discrete alarms
   1: '1UZ1 (A01590) - Привід: перевищено інтервал технічного обслуговування двигуна', class WarningLiftUp, trigger "AlarmsWord1" bit 0
   2: '1UZ1 (A01666) - SI Motion P1 (CU): Постійний сигнал «1» на F-DI для безпечного квитування', class WarningLiftUp, trigger "AlarmsWord1" bit 1
   3: '1UZ1 (A01698) - SI P1 (CU): Активний режим введення в експлуатацію', class WarningLiftUp, trigger "AlarmsWord1" bit 2
   4: '1UZ1 (A01699) - SI P1 (CU): Потрібна тестова зупинка для STO', class WarningLiftUp, trigger "AlarmsWord1" bit 3
   5: '1UZ1 (A01900) - PB/PN: Конфігурація Помилка телеграми', class WarningLiftUp, trigger "AlarmsWord1" bit 4
   6: '1UZ1(A01920) - PROFIBUS: перервано циклічне з’єднання', class WarningLiftUp, trigger "AlarmsWord1" bit 5
   7: '1UZ1 (A05000) - Силовий модуль: перегрів радіатора інвертора AC', class WarningLiftUp, trigger "AlarmsWord1" bit 6
   8: '1UZ1 (A05001) - Силовий модуль: перегрів кристала запірного шару', class WarningLiftUp, trigger "AlarmsWord1" bit 7
   9: '1UZ1 (A05002) - Силовий модуль: перегрів повітря на вході', class WarningLiftUp, trigger "AlarmsWord1" bit 8
   10: '1UZ1 (A05004) - Силовий модуль: перегрів випрямляча', class WarningLiftUp, trigger "AlarmsWord1" bit 9
   11: '1UZ1 (A05006) - Силовий модуль: перегрів за тепловою моделлю', class WarningLiftUp, trigger "AlarmsWord1" bit 10
   12: '1UZ1 (A07012) - Привід: Двигун температура модель 1/3 перегрів', class WarningLiftUp, trigger "AlarmsWord1" bit 11
   13: '1UZ1 (A01013) - CU: Досягнуто або перевищено граничний ресурс вентилятора', class WarningLiftUp, trigger "AlarmsWord1" bit 12
   14: '1UZ1 (A07321) - Привід: Автоматичний перезапуск активний', class WarningLiftUp, trigger "AlarmsWord1" bit 13
   15: '1UZ1 (A07400) - Привід: активний регулятор максимальної напруги кола постійного струму', class WarningLiftUp, trigger "AlarmsWord1" bit 14
   16: '1UZ1 (A07409) - Привід: керування U/f, активний регулятор обмеження струму', class WarningLiftUp, trigger "AlarmsWord1" bit 15
   18: '1UZ1 (A07805) - Ввід: перевантаження I²t силового модуля', class WarningLiftUp, trigger "AlarmsWord2" bit 0
   19: '1UZ1 (A07850) - Зовнішній аварійне повідомлення 1', class WarningLiftUp, trigger "AlarmsWord2" bit 1
   20: '1UZ1 (A07851) - Зовнішній аварійне повідомлення 2', class WarningLiftUp, trigger "AlarmsWord2" bit 2
   21: '1UZ1 (A07852) - Зовнішній аварійне повідомлення 3', class WarningLiftUp, trigger "AlarmsWord2" bit 3
   22: '1UZ1 (A07903) - Привід: відхилення швидкості двигуна', class WarningLiftUp, trigger "AlarmsWord2" bit 4
   23: '1UZ1 (A07910) - Привід: перегрів двигуна', class WarningLiftUp, trigger "AlarmsWord2" bit 5
   24: '1UZ1 (A07920) - Привід: крутний момент/швидкість занадто низькі', class WarningLiftUp, trigger "AlarmsWord2" bit 6
   25: '1UZ1 (A07921) - Привід: крутний момент/швидкість занадто високі', class WarningLiftUp, trigger "AlarmsWord2" bit 7
   26: '1UZ1 (A07922) - Привід: крутний момент/швидкість поза межами допуску', class WarningLiftUp, trigger "AlarmsWord2" bit 8
   27: '1UZ1 (A07927) - DC гальмівний активний', class WarningLiftUp, trigger "AlarmsWord2" bit 9
   28: '1UZ1 (A07980) - Привід: Обертовий вимірювання активовано', class WarningLiftUp, trigger "AlarmsWord2" bit 10
   29: '1UZ1 (A07981) - Привід: Увімкнути сигнали для обертовий вимірювання відсутній', class WarningLiftUp, trigger "AlarmsWord2" bit 11
   30: '1UZ1 (A07991) - Привід: Ідентифікація даних двигуна активовано', class WarningLiftUp, trigger "AlarmsWord2" bit 12
   31: '1UZ1 (A08511) - PN/COMM BOARD: Приймання конфігурація дані некоректний', class WarningLiftUp, trigger "AlarmsWord2" bit 13
   32: '1UZ1 (A08526) - PN/COMM BOARD: Відсутній циклічний з’єднання', class WarningLiftUp, trigger "AlarmsWord2" bit 14
   33: '1UZ1 (A08565) - PNCOMM BOARD: Узгодженість помилка що впливає на регульований параметри', class WarningLiftUp, trigger "AlarmsWord2" bit 15
   35: '1UZ1 (A30049) - Силовий модуль: несправний внутрішній вентилятор', class WarningLiftUp, trigger "AlarmsWord3" bit 0
   36: '1UZ1 (A30502) - Силовий модуль: Перенапруга кола постійного струму', class WarningLiftUp, trigger "AlarmsWord3" bit 1
   37: '1UZ1 (A30920) - Силовий модуль: несправність датчика температури', class WarningLiftUp, trigger "AlarmsWord3" bit 2
   39: '1UZ1 (F01000) - Внутрішня програмна помилка', class ErrorLiftUp, trigger "FaultsWord1" bit 0
   40: '1UZ1 (F01001) - Виняток операції з плаваючою комою', class ErrorLiftUp, trigger "FaultsWord1" bit 1
   41: '1UZ1 (F01015) - Внутрішня програмна помилка', class ErrorLiftUp, trigger "FaultsWord1" bit 2
   42: '1UZ1 (F01033) - Перемикання одиниць: некоректне опорне значення параметра', class ErrorLiftUp, trigger "FaultsWord1" bit 3
   43: '1UZ1 (F01034) - Перемикання одиниць: не вдалося обчислити значення параметрів після зміни опорного значення', class ErrorLiftUp, trigger "FaultsWord1" bit 4
   44: '1UZ1 (F01040) - Збережіть налаштування параметрів і виконайте повторне увімкнення живлення', class ErrorLiftUp, trigger "FaultsWord1" bit 5
   45: '1UZ1 (F01044) - CU: Помилка описових даних', class ErrorLiftUp, trigger "FaultsWord1" bit 6
   46: '1UZ1 (F01054) - CU: Перевищено системне обмеження', class ErrorLiftUp, trigger "FaultsWord1" bit 7
   47: '1UZ1 (F01105) - CU: Недостатньо пам’яті', class ErrorLiftUp, trigger "FaultsWord1" bit 8
   48: '1UZ1 (F01122) - Частота на вході вимірювального щупа занадто висока', class ErrorLiftUp, trigger "FaultsWord1" bit 9
   49: '1UZ1 (F01205) - CU: Переповнення часового кванта', class ErrorLiftUp, trigger "FaultsWord1" bit 10
   50: '1UZ1 (F01250) - CU: Некоректні дані CU-EEPROM, доступні лише для читання', class ErrorLiftUp, trigger "FaultsWord1" bit 11
   51: '1UZ1 (F01512) - BICO: масштабування недоступне', class ErrorLiftUp, trigger "FaultsWord1" bit 12
   52: '1UZ1 (F01600) - SI P1 (CU): Ініційовано зупинку A', class ErrorLiftUp, trigger "FaultsWord1" bit 13
   53: '1UZ1 (F01625) - SI P1 (CU): Помилка сигналу справності в даних безпеки', class ErrorLiftUp, trigger "FaultsWord1" bit 14
   54: '1UZ1 (F01650) - SI P1 (CU): Потрібне приймальне випробування', class ErrorLiftUp, trigger "FaultsWord1" bit 15
   56: '1UZ1 (F01659) - SI P1 (CU): Запит на запис параметра відхилено', class ErrorLiftUp, trigger "FaultsWord2" bit 0
   57: '1UZ1 (F01666) - SI Motion P1 (CU): Постійний сигнал «1» на F-DI для безпечного квитування', class ErrorLiftUp, trigger "FaultsWord2" bit 1
   58: '1UZ1 (F01910) - Польова шина: тайм-аут заданого значення', class ErrorLiftUp, trigger "FaultsWord2" bit 2
   59: '1UZ1 (F06310) - Ввід: напругу живлення (p0210) параметризовано некоректно', class ErrorLiftUp, trigger "FaultsWord2" bit 3
   60: '1UZ1 (F07011) - Привід: перегрів двигуна', class ErrorLiftUp, trigger "FaultsWord2" bit 4
   61: '1UZ1 (F07016) - Привід: Несправність датчика температури двигуна', class ErrorLiftUp, trigger "FaultsWord2" bit 5
   62: '1UZ1 (F07086) - Перемикання одиниць: порушення обмеження параметра через зміну опорного значення', class ErrorLiftUp, trigger "FaultsWord2" bit 6
   63: '1UZ1 (F07088) - Перемикання одиниць: порушення обмеження параметра через перемикання одиниць', class ErrorLiftUp, trigger "FaultsWord2" bit 7
   64: '1UZ1 (F07320) - Привід: Автоматичний перезапуск перервано', class ErrorLiftUp, trigger "FaultsWord2" bit 8
   65: '1UZ1 (F07330) - Підхоплення обертового двигуна: виміряний пошуковий струм занадто малий', class ErrorLiftUp, trigger "FaultsWord2" bit 9
   66: '1UZ1 (F07426) - Технологія регулятор фактичний значення обмежений', class ErrorLiftUp, trigger "FaultsWord2" bit 10
   67: '1UZ1 (F07801) - Привід: Двигун Перевищення струму', class ErrorLiftUp, trigger "FaultsWord2" bit 11
   68: '1UZ1 (F07807) - Привід: виявлено коротке замикання/замикання на землю', class ErrorLiftUp, trigger "FaultsWord2" bit 12
   69: '1UZ1 (F07860) - Зовнішній несправність 1', class ErrorLiftUp, trigger "FaultsWord2" bit 13
   70: '1UZ1 (F07861) - Зовнішній несправність 2', class ErrorLiftUp, trigger "FaultsWord2" bit 14
   71: '1UZ1 (F07862) - Зовнішній несправність 3', class ErrorLiftUp, trigger "FaultsWord2" bit 15
   74: '1UZ1 (F07900) - Привід: заклинювання двигуна/регулятор швидкості на межі', class ErrorLiftUp, trigger "FaultsWord3" bit 0
   75: '1UZ1 (F07901) - Привід: перевищення швидкості двигуна', class ErrorLiftUp, trigger "FaultsWord3" bit 1
   76: '1UZ1 (F07902) - Привід: двигун зупинився', class ErrorLiftUp, trigger "FaultsWord3" bit 2
   77: '1UZ1 (F07923) - Привід: крутний момент/швидкість занадто низькі', class ErrorLiftUp, trigger "FaultsWord3" bit 3
   78: '1UZ1 (F07924) - Привід: крутний момент/швидкість занадто високі', class ErrorLiftUp, trigger "FaultsWord3" bit 4
   79: '1UZ1 (F08501) - PN/COMM BOARD: тайм-аут заданого значення', class ErrorLiftUp, trigger "FaultsWord3" bit 5
   80: '1UZ1 (F08502) - PN/COMM BOARD: закінчився контрольний час сигналу справності', class ErrorLiftUp, trigger "FaultsWord3" bit 6
   81: '1UZ1 (F06210) - Ввід: Сумування струм занадто високий', class ErrorLiftUp, trigger "FaultsWord3" bit 7
   82: '1UZ1 (F13100) - Захист ноу-хау: помилка захисту від копіювання', class ErrorLiftUp, trigger "FaultsWord3" bit 8
   83: '1UZ1 (F13101) - Захист ноу-хау: неможливо активувати захист від копіювання', class ErrorLiftUp, trigger "FaultsWord3" bit 9
   84: '1UZ1 (F30001) - Силовий модуль: перевищення струму', class ErrorLiftUp, trigger "FaultsWord3" bit 10
   85: '1UZ1 (F30002) - Силовий модуль: перенапруга кола постійного струму', class ErrorLiftUp, trigger "FaultsWord3" bit 11
   86: '1UZ1 (F30003) - Силовий модуль: занижена напруга кола постійного струму', class ErrorLiftUp, trigger "FaultsWord3" bit 12
   87: '1UZ1 (F30004) - Силовий модуль: перегрів радіатора інвертора AC', class ErrorLiftUp, trigger "FaultsWord3" bit 13
   88: '1UZ1 (F30005) - Силовий модуль: перевантаження I²t', class ErrorLiftUp, trigger "FaultsWord3" bit 14
   89: '1UZ1 (F30011) - Силовий модуль: відсутня фаза мережі в головному колі', class ErrorLiftUp, trigger "FaultsWord3" bit 15
   91: '1UZ1 (F30015) - Силовий модуль: відсутня фаза кабелю двигуна', class ErrorLiftUp, trigger "FaultsWord4" bit 0
   92: '1UZ1 (F30021) - Силовий модуль: замикання на землю', class ErrorLiftUp, trigger "FaultsWord4" bit 1
   93: '1UZ1 (F30022) - Силовий модуль: контроль Uce', class ErrorLiftUp, trigger "FaultsWord4" bit 2
   94: '1UZ1 (F30027) - Силовий модуль: контроль часу попереднього заряду кола постійного струму', class ErrorLiftUp, trigger "FaultsWord4" bit 3
   95: '1UZ1 (F30035) - Силовий модуль: перегрів повітря на вході', class ErrorLiftUp, trigger "FaultsWord4" bit 4
   96: '1UZ1 (F30036) - Силовий модуль: внутрішній перегрів', class ErrorLiftUp, trigger "FaultsWord4" bit 5
   97: '1UZ1 (F30037) - Силовий модуль: перегрів випрямляча', class ErrorLiftUp, trigger "FaultsWord4" bit 6
   98: '1UZ1 (F30052) - Помилка даних EEPROM', class ErrorLiftUp, trigger "FaultsWord4" bit 7
   99: '1UZ1 (F30053) - FPGA дані несправний', class ErrorLiftUp, trigger "FaultsWord4" bit 8
   100: '1UZ1 (F30059) - Силовий модуль: несправний внутрішній вентилятор', class ErrorLiftUp, trigger "FaultsWord4" bit 9
   101: '1UZ1 (F30074) - Помилка зв’язку між Керування Модуль та Силовий модуль', class ErrorLiftUp, trigger "FaultsWord4" bit 10
   102: '1UZ1 (F30600) - SI P2: Ініційовано зупинку A', class ErrorLiftUp, trigger "FaultsWord4" bit 11
   103: '1UZ1 (F30664) - Помилка під час завантаження', class ErrorLiftUp, trigger "FaultsWord4" bit 12
   104: '1UZ1 (F30850) - Силовий модуль: Внутрішня програмна помилка', class ErrorLiftUp, trigger "FaultsWord4" bit 13
   38: '1UZ1 (F06211) - Ввід: сумарний струм неприпустимо високий', class ErrorLiftUp, trigger "FaultsWord4" bit 14
   105: '1UZ1 (F08510) - PN/COMM BOARD: некоректні дані конфігурації передавання', class ErrorLiftUp, trigger "FaultsWord4" bit 15
   106: '3UZ1 (A01590) - Привід: перевищено інтервал технічного обслуговування двигуна', class WarningTrolley, trigger "AlarmsWord1" bit 0
   107: '3UZ1 (A01666) - SI Motion P1 (CU): Постійний сигнал «1» на F-DI для безпечного квитування', class WarningTrolley, trigger "AlarmsWord1" bit 1
   108: '3UZ1 (A01698) - SI P1 (CU): Активний режим введення в експлуатацію', class WarningTrolley, trigger "AlarmsWord1" bit 2
   109: '3UZ1 (A01699) - SI P1 (CU): Потрібна тестова зупинка для STO', class WarningTrolley, trigger "AlarmsWord1" bit 3
   110: '3UZ1 (A01900) - PB/PN: Конфігурація Помилка телеграми', class WarningTrolley, trigger "AlarmsWord1" bit 4
   111: '3UZ1(A01920) - PROFIBUS: перервано циклічне з’єднання', class WarningTrolley, trigger "AlarmsWord1" bit 5
   112: '3UZ1 (A05000) - Силовий модуль: перегрів радіатора інвертора AC', class WarningTrolley, trigger "AlarmsWord1" bit 6
   113: '3UZ1 (A05001) - Силовий модуль: перегрів кристала запірного шару', class WarningTrolley, trigger "AlarmsWord1" bit 7
   114: '3UZ1 (A05002) - Силовий модуль: перегрів повітря на вході', class WarningTrolley, trigger "AlarmsWord1" bit 8
   115: '3UZ1 (A05004) - Силовий модуль: перегрів випрямляча', class WarningTrolley, trigger "AlarmsWord1" bit 9
   116: '3UZ1 (A05006) - Силовий модуль: перегрів за тепловою моделлю', class WarningTrolley, trigger "AlarmsWord1" bit 10
   117: '3UZ1 (A07012) - Привід: Двигун температура модель 1/3 перегрів', class WarningTrolley, trigger "AlarmsWord1" bit 11
   118: '3UZ1 (A01013) - CU: Досягнуто або перевищено граничний ресурс вентилятора', class WarningTrolley, trigger "AlarmsWord1" bit 12
   119: '3UZ1 (A07321) - Привід: Автоматичний перезапуск активний', class WarningTrolley, trigger "AlarmsWord1" bit 13
   120: '3UZ1 (A07400) - Привід: активний регулятор максимальної напруги кола постійного струму', class WarningTrolley, trigger "AlarmsWord1" bit 14
   121: '3UZ1 (A07409) - Привід: керування U/f, активний регулятор обмеження струму', class WarningTrolley, trigger "AlarmsWord1" bit 15
   122: '3UZ1 (A07805) - Ввід: перевантаження I²t силового модуля', class WarningTrolley, trigger "AlarmsWord2" bit 0
   123: '3UZ1 (A07850) - Зовнішній аварійне повідомлення 1', class WarningTrolley, trigger "AlarmsWord2" bit 1
   124: '3UZ1 (A07851) - Зовнішній аварійне повідомлення 2', class WarningTrolley, trigger "AlarmsWord2" bit 2
   125: '3UZ1 (A07852) - Зовнішній аварійне повідомлення 3', class WarningTrolley, trigger "AlarmsWord2" bit 3
   126: '3UZ1 (A07903) - Привід: відхилення швидкості двигуна', class WarningTrolley, trigger "AlarmsWord2" bit 4
   127: '3UZ1 (A07910) - Привід: перегрів двигуна', class WarningTrolley, trigger "AlarmsWord2" bit 5
   128: '3UZ1 (A07920) - Привід: крутний момент/швидкість занадто низькі', class WarningTrolley, trigger "AlarmsWord2" bit 6
   129: '3UZ1 (A07921) - Привід: крутний момент/швидкість занадто високі', class WarningTrolley, trigger "AlarmsWord2" bit 7
   130: '3UZ1 (A07922) - Привід: крутний момент/швидкість поза межами допуску', class WarningTrolley, trigger "AlarmsWord2" bit 8
   131: '3UZ1 (A07927) - DC гальмівний активний', class WarningTrolley, trigger "AlarmsWord2" bit 9
   132: '3UZ1 (A07980) - Привід: Обертовий вимірювання активовано', class WarningTrolley, trigger "AlarmsWord2" bit 10
   133: '3UZ1 (A07981) - Привід: Увімкнути сигнали для обертовий вимірювання відсутній', class WarningTrolley, trigger "AlarmsWord2" bit 11
   134: '3UZ1 (A07991) - Привід: Ідентифікація даних двигуна активовано', class WarningTrolley, trigger "AlarmsWord2" bit 12
   135: '3UZ1 (A08511) - PN/COMM BOARD: Приймання конфігурація дані некоректний', class WarningTrolley, trigger "AlarmsWord2" bit 13
   136: '3UZ1 (A08526) - PN/COMM BOARD: Відсутній циклічний з’єднання', class WarningTrolley, trigger "AlarmsWord2" bit 14
   137: '3UZ1 (A08565) - PNCOMM BOARD: Узгодженість помилка що впливає на регульований параметри', class WarningTrolley, trigger "AlarmsWord2" bit 15
   138: '3UZ1 (A30049) - Силовий модуль: несправний внутрішній вентилятор', class WarningTrolley, trigger "AlarmsWord3" bit 0
   139: '3UZ1 (A30502) - Силовий модуль: Перенапруга кола постійного струму', class WarningTrolley, trigger "AlarmsWord3" bit 1
   140: '3UZ1 (A30920) - Силовий модуль: несправність датчика температури', class WarningTrolley, trigger "AlarmsWord3" bit 2
   141: '3UZ1 (F01000) - Внутрішня програмна помилка', class ErrorTrolley, trigger "FaultsWord1" bit 0
   142: '3UZ1 (F01001) - Виняток операції з плаваючою комою', class ErrorTrolley, trigger "FaultsWord1" bit 1
   143: '3UZ1 (F01015) - Внутрішня програмна помилка', class ErrorTrolley, trigger "FaultsWord1" bit 2
   144: '3UZ1 (F01033) - Перемикання одиниць: некоректне опорне значення параметра', class ErrorTrolley, trigger "FaultsWord1" bit 3
   145: '3UZ1 (F01034) - Перемикання одиниць: не вдалося обчислити значення параметрів після зміни опорного значення', class ErrorTrolley, trigger "FaultsWord1" bit 4
   146: '3UZ1 (F01040) - Збережіть налаштування параметрів і виконайте повторне увімкнення живлення', class ErrorTrolley, trigger "FaultsWord1" bit 5
   147: '3UZ1 (F01044) - CU: Помилка описових даних', class ErrorTrolley, trigger "FaultsWord1" bit 6
   148: '3UZ1 (F01054) - CU: Перевищено системне обмеження', class ErrorTrolley, trigger "FaultsWord1" bit 7
   149: '3UZ1 (F01105) - CU: Недостатньо пам’яті', class ErrorTrolley, trigger "FaultsWord1" bit 8
   150: '3UZ1 (F01122) - Частота на вході вимірювального щупа занадто висока', class ErrorTrolley, trigger "FaultsWord1" bit 9
   151: '3UZ1 (F01205) - CU: Переповнення часового кванта', class ErrorTrolley, trigger "FaultsWord1" bit 10
   152: '3UZ1 (F01250) - CU: Некоректні дані CU-EEPROM, доступні лише для читання', class ErrorTrolley, trigger "FaultsWord1" bit 11
   153: '3UZ1 (F01512) - BICO: масштабування недоступне', class ErrorTrolley, trigger "FaultsWord1" bit 12
   154: '3UZ1 (F01600) - SI P1 (CU): Ініційовано зупинку A', class ErrorTrolley, trigger "FaultsWord1" bit 13
   155: '3UZ1 (F01625) - SI P1 (CU): Помилка сигналу справності в даних безпеки', class ErrorTrolley, trigger "FaultsWord1" bit 14
   156: '3UZ1 (F01650) - SI P1 (CU): Потрібне приймальне випробування', class ErrorTrolley, trigger "FaultsWord1" bit 15
   157: '3UZ1 (F01659) - SI P1 (CU): Запит на запис параметра відхилено', class ErrorTrolley, trigger "FaultsWord2" bit 0
   158: '3UZ1 (F01666) - SI Motion P1 (CU): Постійний сигнал «1» на F-DI для безпечного квитування', class ErrorTrolley, trigger "FaultsWord2" bit 1
   159: '3UZ1 (F01910) - Польова шина: тайм-аут заданого значення', class ErrorTrolley, trigger "FaultsWord2" bit 2
   160: '3UZ1 (F06310) - Ввід: напругу живлення (p0210) параметризовано некоректно', class ErrorTrolley, trigger "FaultsWord2" bit 3
   161: '3UZ1 (F07011) - Привід: перегрів двигуна', class ErrorTrolley, trigger "FaultsWord2" bit 4
   162: '3UZ1 (F07016) - Привід: Несправність датчика температури двигуна', class ErrorTrolley, trigger "FaultsWord2" bit 5
   163: '3UZ1 (F07086) - Перемикання одиниць: порушення обмеження параметра через зміну опорного значення', class ErrorTrolley, trigger "FaultsWord2" bit 6
   164: '3UZ1 (F07088) - Перемикання одиниць: порушення обмеження параметра через перемикання одиниць', class ErrorTrolley, trigger "FaultsWord2" bit 7
   165: '3UZ1 (F07320) - Привід: Автоматичний перезапуск перервано', class ErrorTrolley, trigger "FaultsWord2" bit 8
   166: '3UZ1 (F07330) - Підхоплення обертового двигуна: виміряний пошуковий струм занадто малий', class ErrorTrolley, trigger "FaultsWord2" bit 9
   167: '3UZ1 (F07426) - Технологія регулятор фактичний значення обмежений', class ErrorTrolley, trigger "FaultsWord2" bit 10
   168: '3UZ1 (F07801) - Привід: Двигун Перевищення струму', class ErrorTrolley, trigger "FaultsWord2" bit 11
   169: '3UZ1 (F07807) - Привід: виявлено коротке замикання/замикання на землю', class ErrorTrolley, trigger "FaultsWord2" bit 12
   170: '3UZ1 (F07860) - Зовнішній несправність 1', class ErrorTrolley, trigger "FaultsWord2" bit 13
   171: '3UZ1 (F07861) - Зовнішній несправність 2', class ErrorTrolley, trigger "FaultsWord2" bit 14
   172: '3UZ1 (F07862) - Зовнішній несправність 3', class ErrorTrolley, trigger "FaultsWord2" bit 15
   173: '3UZ1 (F07900) - Привід: заклинювання двигуна/регулятор швидкості на межі', class ErrorTrolley, trigger "FaultsWord3" bit 0
   174: '3UZ1 (F07901) - Привід: перевищення швидкості двигуна', class ErrorTrolley, trigger "FaultsWord3" bit 1
   175: '3UZ1 (F07902) - Привід: двигун зупинився', class ErrorTrolley, trigger "FaultsWord3" bit 2
   176: '3UZ1 (F07923) - Привід: крутний момент/швидкість занадто низькі', class ErrorTrolley, trigger "FaultsWord3" bit 3
   177: '3UZ1 (F07924) - Привід: крутний момент/швидкість занадто високі', class ErrorTrolley, trigger "FaultsWord3" bit 4
   178: '3UZ1 (F08501) - PN/COMM BOARD: тайм-аут заданого значення', class ErrorTrolley, trigger "FaultsWord3" bit 5
   179: '3UZ1 (F08502) - PN/COMM BOARD: закінчився контрольний час сигналу справності', class ErrorTrolley, trigger "FaultsWord3" bit 6
   180: '3UZ1 (F06210) - Ввід: Сумування струм занадто високий', class ErrorTrolley, trigger "FaultsWord3" bit 7
   181: '3UZ1 (F13100) - Захист ноу-хау: помилка захисту від копіювання', class ErrorTrolley, trigger "FaultsWord3" bit 8
   182: '3UZ1 (F13101) - Захист ноу-хау: неможливо активувати захист від копіювання', class ErrorTrolley, trigger "FaultsWord3" bit 9
   183: '3UZ1 (F30001) - Силовий модуль: перевищення струму', class ErrorTrolley, trigger "FaultsWord3" bit 10
   184: '3UZ1 (F30002) - Силовий модуль: перенапруга кола постійного струму', class ErrorTrolley, trigger "FaultsWord3" bit 11
   185: '3UZ1 (F30003) - Силовий модуль: занижена напруга кола постійного струму', class ErrorTrolley, trigger "FaultsWord3" bit 12
   186: '3UZ1 (F30004) - Силовий модуль: перегрів радіатора інвертора AC', class ErrorTrolley, trigger "FaultsWord3" bit 13
   187: '3UZ1 (F30005) - Силовий модуль: перевантаження I²t', class ErrorTrolley, trigger "FaultsWord3" bit 14
   188: '3UZ1 (F30011) - Силовий модуль: відсутня фаза мережі в головному колі', class ErrorTrolley, trigger "FaultsWord3" bit 15
   189: '3UZ1 (F30015) - Силовий модуль: відсутня фаза кабелю двигуна', class ErrorTrolley, trigger "FaultsWord4" bit 0
   190: '3UZ1 (F30021) - Силовий модуль: замикання на землю', class ErrorTrolley, trigger "FaultsWord4" bit 1
   191: '3UZ1 (F30022) - Силовий модуль: контроль Uce', class ErrorTrolley, trigger "FaultsWord4" bit 2
   192: '3UZ1 (F30027) - Силовий модуль: контроль часу попереднього заряду кола постійного струму', class ErrorTrolley, trigger "FaultsWord4" bit 3
   193: '3UZ1 (F30035) - Силовий модуль: перегрів повітря на вході', class ErrorTrolley, trigger "FaultsWord4" bit 4
   194: '3UZ1 (F30036) - Силовий модуль: внутрішній перегрів', class ErrorTrolley, trigger "FaultsWord4" bit 5
   195: '3UZ1 (F30037) - Силовий модуль: перегрів випрямляча', class ErrorTrolley, trigger "FaultsWord4" bit 6
   196: '3UZ1 (F30052) - Помилка даних EEPROM', class ErrorTrolley, trigger "FaultsWord4" bit 7
   197: '3UZ1 (F30053) - FPGA дані несправний', class ErrorTrolley, trigger "FaultsWord4" bit 8
   198: '3UZ1 (F30059) - Силовий модуль: несправний внутрішній вентилятор', class ErrorTrolley, trigger "FaultsWord4" bit 9
   199: '3UZ1 (F30074) - Помилка зв’язку між Керування Модуль та Силовий модуль', class ErrorTrolley, trigger "FaultsWord4" bit 10
   200: '3UZ1 (F30600) - SI P2: Ініційовано зупинку A', class ErrorTrolley, trigger "FaultsWord4" bit 11
   201: '3UZ1 (F30664) - Помилка під час завантаження', class ErrorTrolley, trigger "FaultsWord4" bit 12
   202: '3UZ1 (F30850) - Силовий модуль: Внутрішня програмна помилка', class ErrorTrolley, trigger "FaultsWord4" bit 13
   203: '3UZ1 (F06211) - Ввід: сумарний струм неприпустимо високий', class ErrorTrolley, trigger "FaultsWord4" bit 14
   204: '3UZ1 (F08510) - PN/COMM BOARD: некоректні дані конфігурації передавання', class ErrorTrolley, trigger "FaultsWord4" bit 15
   205: '4UZ1 (A01590) - Привід: перевищено інтервал технічного обслуговування двигуна', class WarningCrane, trigger "AlarmsWord1" bit 0
   206: '4UZ1 (A01666) - SI Motion P1 (CU): Постійний сигнал «1» на F-DI для безпечного квитування', class WarningCrane, trigger "AlarmsWord1" bit 1
   207: '4UZ1 (A01698) - SI P1 (CU): Активний режим введення в експлуатацію', class WarningCrane, trigger "AlarmsWord1" bit 2
   208: '4UZ1 (A01699) - SI P1 (CU): Потрібна тестова зупинка для STO', class WarningCrane, trigger "AlarmsWord1" bit 3
   209: '4UZ1 (A01900) - PB/PN: Конфігурація Помилка телеграми', class WarningCrane, trigger "AlarmsWord1" bit 4
   210: '4UZ1(A01920) - PROFIBUS: перервано циклічне з’єднання', class WarningCrane, trigger "AlarmsWord1" bit 5
   211: '4UZ1 (A05000) - Силовий модуль: перегрів радіатора інвертора AC', class WarningCrane, trigger "AlarmsWord1" bit 6
   212: '4UZ1 (A05001) - Силовий модуль: перегрів кристала запірного шару', class WarningCrane, trigger "AlarmsWord1" bit 7
   213: '4UZ1 (A05002) - Силовий модуль: перегрів повітря на вході', class WarningCrane, trigger "AlarmsWord1" bit 8
   214: '4UZ1 (A05004) - Силовий модуль: перегрів випрямляча', class WarningCrane, trigger "AlarmsWord1" bit 9
   215: '4UZ1 (A05006) - Силовий модуль: перегрів за тепловою моделлю', class WarningCrane, trigger "AlarmsWord1" bit 10
   216: '4UZ1 (A07012) - Привід: Двигун температура модель 1/3 перегрів', class WarningCrane, trigger "AlarmsWord1" bit 11
   217: '4UZ1 (A01013) - CU: Досягнуто або перевищено граничний ресурс вентилятора', class WarningCrane, trigger "AlarmsWord1" bit 12
   218: '4UZ1 (A07321) - Привід: Автоматичний перезапуск активний', class WarningCrane, trigger "AlarmsWord1" bit 13
   219: '4UZ1 (A07400) - Привід: активний регулятор максимальної напруги кола постійного струму', class WarningCrane, trigger "AlarmsWord1" bit 14
   220: '4UZ1 (A07409) - Привід: керування U/f, активний регулятор обмеження струму', class WarningCrane, trigger "AlarmsWord1" bit 15
   221: '4UZ1 (A07805) - Ввід: перевантаження I²t силового модуля', class WarningCrane, trigger "AlarmsWord2" bit 0
   222: '4UZ1 (A07850) - Зовнішній аварійне повідомлення 1', class WarningCrane, trigger "AlarmsWord2" bit 1
   223: '4UZ1 (A07851) - Зовнішній аварійне повідомлення 2', class WarningCrane, trigger "AlarmsWord2" bit 2
   224: '4UZ1 (A07852) - Зовнішній аварійне повідомлення 3', class WarningCrane, trigger "AlarmsWord2" bit 3
   225: '4UZ1 (A07903) - Привід: відхилення швидкості двигуна', class WarningCrane, trigger "AlarmsWord2" bit 4
   226: '4UZ1 (A07910) - Привід: перегрів двигуна', class WarningCrane, trigger "AlarmsWord2" bit 5
   227: '4UZ1 (A07920) - Привід: крутний момент/швидкість занадто низькі', class WarningCrane, trigger "AlarmsWord2" bit 6
   228: '4UZ1 (A07921) - Привід: крутний момент/швидкість занадто високі', class WarningCrane, trigger "AlarmsWord2" bit 7
   229: '4UZ1 (A07922) - Привід: крутний момент/швидкість поза межами допуску', class WarningCrane, trigger "AlarmsWord2" bit 8
   230: '4UZ1 (A07927) - DC гальмівний активний', class WarningCrane, trigger "AlarmsWord2" bit 9
   231: '4UZ1 (A07980) - Привід: Обертовий вимірювання активовано', class WarningCrane, trigger "AlarmsWord2" bit 10
   232: '4UZ1 (A07981) - Привід: Увімкнути сигнали для обертовий вимірювання відсутній', class WarningCrane, trigger "AlarmsWord2" bit 11
   233: '4UZ1 (A07991) - Привід: Ідентифікація даних двигуна активовано', class WarningCrane, trigger "AlarmsWord2" bit 12
   234: '4UZ1 (A08511) - PN/COMM BOARD: Приймання конфігурація дані некоректний', class WarningCrane, trigger "AlarmsWord2" bit 13
   235: '4UZ1 (A08526) - PN/COMM BOARD: Відсутній циклічний з’єднання', class WarningCrane, trigger "AlarmsWord2" bit 14
   236: '4UZ1 (A08565) - PNCOMM BOARD: Узгодженість помилка що впливає на регульований параметри', class WarningCrane, trigger "AlarmsWord2" bit 15
   237: '4UZ1 (A30049) - Силовий модуль: несправний внутрішній вентилятор', class WarningCrane, trigger "AlarmsWord3" bit 0
   238: '4UZ1 (A30502) - Силовий модуль: Перенапруга кола постійного струму', class WarningCrane, trigger "AlarmsWord3" bit 1
   239: '4UZ1 (A30920) - Силовий модуль: несправність датчика температури', class WarningCrane, trigger "AlarmsWord3" bit 2
   240: '4UZ1 (F01000) - Внутрішня програмна помилка', class ErrorCrane, trigger "FaultsWord1" bit 0
   241: '4UZ1 (F01001) - Виняток операції з плаваючою комою', class ErrorCrane, trigger "FaultsWord1" bit 1
   242: '4UZ1 (F01015) - Внутрішня програмна помилка', class ErrorCrane, trigger "FaultsWord1" bit 2
   243: '4UZ1 (F01033) - Перемикання одиниць: некоректне опорне значення параметра', class ErrorCrane, trigger "FaultsWord1" bit 3
   244: '4UZ1 (F01034) - Перемикання одиниць: не вдалося обчислити значення параметрів після зміни опорного значення', class ErrorCrane, trigger "FaultsWord1" bit 4
   245: '4UZ1 (F01040) - Збережіть налаштування параметрів і виконайте повторне увімкнення живлення', class ErrorCrane, trigger "FaultsWord1" bit 5
   246: '4UZ1 (F01044) - CU: Помилка описових даних', class ErrorCrane, trigger "FaultsWord1" bit 6
   247: '4UZ1 (F01054) - CU: Перевищено системне обмеження', class ErrorCrane, trigger "FaultsWord1" bit 7
   248: '4UZ1 (F01105) - CU: Недостатньо пам’яті', class ErrorCrane, trigger "FaultsWord1" bit 8
   249: '4UZ1 (F01122) - Частота на вході вимірювального щупа занадто висока', class ErrorCrane, trigger "FaultsWord1" bit 9
   250: '4UZ1 (F01205) - CU: Переповнення часового кванта', class ErrorCrane, trigger "FaultsWord1" bit 10
   251: '4UZ1 (F01250) - CU: Некоректні дані CU-EEPROM, доступні лише для читання', class ErrorCrane, trigger "FaultsWord1" bit 11
   252: '4UZ1 (F01512) - BICO: масштабування недоступне', class ErrorCrane, trigger "FaultsWord1" bit 12
   253: '4UZ1 (F01600) - SI P1 (CU): Ініційовано зупинку A', class ErrorCrane, trigger "FaultsWord1" bit 13
   254: '4UZ1 (F01625) - SI P1 (CU): Помилка сигналу справності в даних безпеки', class ErrorCrane, trigger "FaultsWord1" bit 14
   255: '4UZ1 (F01650) - SI P1 (CU): Потрібне приймальне випробування', class ErrorCrane, trigger "FaultsWord1" bit 15
   256: '4UZ1 (F01659) - SI P1 (CU): Запит на запис параметра відхилено', class ErrorCrane, trigger "FaultsWord2" bit 0
   257: '4UZ1 (F01666) - SI Motion P1 (CU): Постійний сигнал «1» на F-DI для безпечного квитування', class ErrorCrane, trigger "FaultsWord2" bit 1
   258: '4UZ1 (F01910) - Польова шина: тайм-аут заданого значення', class ErrorCrane, trigger "FaultsWord2" bit 2
   259: '4UZ1 (F01910) - Ввід: напругу живлення (p0210) параметризовано некоректно', class ErrorCrane, trigger "FaultsWord2" bit 3
   260: '4UZ1 (F07011) - Привід: перегрів двигуна', class ErrorCrane, trigger "FaultsWord2" bit 4
   261: '4UZ1 (F07016) - Привід: Несправність датчика температури двигуна', class ErrorCrane, trigger "FaultsWord2" bit 5
   262: '4UZ1 (F07086) - Перемикання одиниць: порушення обмеження параметра через зміну опорного значення', class ErrorCrane, trigger "FaultsWord2" bit 6
   263: '4UZ1 (F07088) - Перемикання одиниць: порушення обмеження параметра через перемикання одиниць', class ErrorCrane, trigger "FaultsWord2" bit 7
   264: '4UZ1 (F07320) - Привід: Автоматичний перезапуск перервано', class ErrorCrane, trigger "FaultsWord2" bit 8
   265: '4UZ1 (F07330) - Підхоплення обертового двигуна: виміряний пошуковий струм занадто малий', class ErrorCrane, trigger "FaultsWord2" bit 9
   266: '4UZ1 (F07426) - Технологія регулятор фактичний значення обмежений', class ErrorCrane, trigger "FaultsWord2" bit 10
   267: '4UZ1 (F07801) - Привід: Двигун Перевищення струму', class ErrorCrane, trigger "FaultsWord2" bit 11
   268: '4UZ1 (F07801) - Привід: виявлено коротке замикання/замикання на землю', class ErrorCrane, trigger "FaultsWord2" bit 12
   269: '4UZ1 (F07860) - Зовнішній несправність 1', class ErrorCrane, trigger "FaultsWord2" bit 13
   270: '4UZ1 (F07861) - Зовнішній несправність 2', class ErrorCrane, trigger "FaultsWord2" bit 14
   271: '4UZ1 (F07861) - Зовнішній несправність 3', class ErrorCrane, trigger "FaultsWord2" bit 15
   272: '4UZ1 (F07900) - Привід: заклинювання двигуна/регулятор швидкості на межі', class ErrorCrane, trigger "FaultsWord3" bit 0
   273: '4UZ1 (F07901) - Привід: перевищення швидкості двигуна', class ErrorCrane, trigger "FaultsWord3" bit 1
   274: '4UZ1 (F07902) - Привід: двигун зупинився', class ErrorCrane, trigger "FaultsWord3" bit 2
   275: '4UZ1 (F07923) - Привід: крутний момент/швидкість занадто низькі', class ErrorCrane, trigger "FaultsWord3" bit 3
   276: '4UZ1 (F07924) - Привід: крутний момент/швидкість занадто високі', class ErrorCrane, trigger "FaultsWord3" bit 4
   277: '4UZ1 (F08501) - PN/COMM BOARD: тайм-аут заданого значення', class ErrorCrane, trigger "FaultsWord3" bit 5
   278: '4UZ1 (F08502) - PN/COMM BOARD: закінчився контрольний час сигналу справності', class ErrorCrane, trigger "FaultsWord3" bit 6
   279: '4UZ1 (F06210) - Ввід: Сумування струм занадто високий', class ErrorCrane, trigger "FaultsWord3" bit 7
   280: '4UZ1 (F13100) - Захист ноу-хау: помилка захисту від копіювання', class ErrorCrane, trigger "FaultsWord3" bit 8
   281: '4UZ1 (F13101) - Захист ноу-хау: неможливо активувати захист від копіювання', class ErrorCrane, trigger "FaultsWord3" bit 9
   282: '4UZ1 (F30001) - Силовий модуль: перевищення струму', class ErrorCrane, trigger "FaultsWord3" bit 10
   283: '4UZ1 (F30002) - Силовий модуль: перенапруга кола постійного струму', class ErrorCrane, trigger "FaultsWord3" bit 11
   284: '4UZ1 (F30003) - Силовий модуль: занижена напруга кола постійного струму', class ErrorCrane, trigger "FaultsWord3" bit 12
   285: '4UZ1 (F30004) - Силовий модуль: перегрів радіатора інвертора AC', class ErrorCrane, trigger "FaultsWord3" bit 13
   286: '4UZ1 (F30005) - Силовий модуль: перевантаження I²t', class ErrorCrane, trigger "FaultsWord3" bit 14
   287: '4UZ1 (F30011) - Силовий модуль: відсутня фаза мережі в головному колі', class ErrorCrane, trigger "FaultsWord3" bit 15
   288: '4UZ1 (F30015) - Силовий модуль: відсутня фаза кабелю двигуна', class ErrorCrane, trigger "FaultsWord4" bit 0
   289: '4UZ1 (F30021) - Силовий модуль: замикання на землю', class ErrorCrane, trigger "FaultsWord4" bit 1
   290: '4UZ1 (F30022) - Силовий модуль: контроль Uce', class ErrorCrane, trigger "FaultsWord4" bit 2
   291: '4UZ1 (F30027) - Силовий модуль: контроль часу попереднього заряду кола постійного струму', class ErrorCrane, trigger "FaultsWord4" bit 3
   292: '4UZ1 (F30035) - Силовий модуль: перегрів повітря на вході', class ErrorCrane, trigger "FaultsWord4" bit 4
   293: '4UZ1 (F30036) - Силовий модуль: внутрішній перегрів', class ErrorCrane, trigger "FaultsWord4" bit 5
   294: '4UZ1 (F30037) - Силовий модуль: перегрів випрямляча', class ErrorCrane, trigger "FaultsWord4" bit 6
   295: '4UZ1 (F30052) - Помилка даних EEPROM', class ErrorCrane, trigger "FaultsWord4" bit 7
   296: '4UZ1 (F30053) - FPGA дані несправний', class ErrorCrane, trigger "FaultsWord4" bit 8
   297: '4UZ1 (F30059) - Силовий модуль: несправний внутрішній вентилятор', class ErrorCrane, trigger "FaultsWord4" bit 9
   298: '4UZ1 (F30074) - Помилка зв’язку між Керування Модуль та Силовий модуль', class ErrorCrane, trigger "FaultsWord4" bit 10
   299: '4UZ1 (F30600) - SI P2: Ініційовано зупинку A', class ErrorCrane, trigger "FaultsWord4" bit 11
   300: '4UZ1 (F30664) - Помилка під час завантаження', class ErrorCrane, trigger "FaultsWord4" bit 12
   301: '4UZ1 (F30850) - Силовий модуль: Внутрішня програмна помилка', class ErrorCrane, trigger "FaultsWord4" bit 13
   302: '4UZ1 (F06211) - Ввід: сумарний струм неприпустимо високий', class ErrorCrane, trigger "FaultsWord4" bit 14
   303: '4UZ1 (F08510) - PN/COMM BOARD: некоректні дані конфігурації передавання', class ErrorCrane, trigger "FaultsWord4" bit 15
   304: '4UZ2 (A01590) - Привід: перевищено інтервал технічного обслуговування двигуна', class WarningCrane, trigger "AlarmsWord1" bit 0
   305: '4UZ2 (A01666) - SI Motion P1 (CU): Постійний сигнал «1» на F-DI для безпечного квитування', class WarningCrane, trigger "AlarmsWord1" bit 1
   306: '4UZ2 (A01698) - SI P1 (CU): Активний режим введення в експлуатацію', class WarningCrane, trigger "AlarmsWord1" bit 2
   307: '4UZ2 (A01699) - SI P1 (CU): Потрібна тестова зупинка для STO', class WarningCrane, trigger "AlarmsWord1" bit 3
   308: '4UZ2 (A01900) - PB/PN: Конфігурація Помилка телеграми', class WarningCrane, trigger "AlarmsWord1" bit 4
   309: '4UZ2(A01920) - PROFIBUS: перервано циклічне з’єднання', class WarningCrane, trigger "AlarmsWord1" bit 5
   310: '4UZ2 (A05000) - Силовий модуль: перегрів радіатора інвертора AC', class WarningCrane, trigger "AlarmsWord1" bit 6
   311: '4UZ2 (A05001) - Силовий модуль: перегрів кристала запірного шару', class WarningCrane, trigger "AlarmsWord1" bit 7
   312: '4UZ2 (A05002) - Силовий модуль: перегрів повітря на вході', class WarningCrane, trigger "AlarmsWord1" bit 8
   313: '4UZ2 (A05004) - Силовий модуль: перегрів випрямляча', class WarningCrane, trigger "AlarmsWord1" bit 9
   314: '4UZ2 (A05006) - Силовий модуль: перегрів за тепловою моделлю', class WarningCrane, trigger "AlarmsWord1" bit 10
   315: '4UZ2 (A07012) - Привід: Двигун температура модель 1/3 перегрів', class WarningCrane, trigger "AlarmsWord1" bit 11
   316: '4UZ2 (A01013) - CU: Досягнуто або перевищено граничний ресурс вентилятора', class WarningCrane, trigger "AlarmsWord1" bit 12
   317: '4UZ2 (A07321) - Привід: Автоматичний перезапуск активний', class WarningCrane, trigger "AlarmsWord1" bit 13
   318: '4UZ2 (A07400) - Привід: активний регулятор максимальної напруги кола постійного струму', class WarningCrane, trigger "AlarmsWord1" bit 14
   319: '4UZ2 (A07409) - Привід: керування U/f, активний регулятор обмеження струму', class WarningCrane, trigger "AlarmsWord1" bit 15
   320: '4UZ2 (A07805) - Ввід: перевантаження I²t силового модуля', class WarningCrane, trigger "AlarmsWord2" bit 0
   321: '4UZ2 (A07850) - Зовнішній аварійне повідомлення 1', class WarningCrane, trigger "AlarmsWord2" bit 1
   322: '4UZ2 (A07851) - Зовнішній аварійне повідомлення 2', class WarningCrane, trigger "AlarmsWord2" bit 2
   323: '4UZ2 (A07852) - Зовнішній аварійне повідомлення 3', class WarningCrane, trigger "AlarmsWord2" bit 3
   324: '4UZ2 (A07903) - Привід: відхилення швидкості двигуна', class WarningCrane, trigger "AlarmsWord2" bit 4
   325: '4UZ2 (A07910) - Привід: перегрів двигуна', class WarningCrane, trigger "AlarmsWord2" bit 5
   326: '4UZ2 (A07920) - Привід: крутний момент/швидкість занадто низькі', class WarningCrane, trigger "AlarmsWord2" bit 6
   327: '4UZ2 (A07921) - Привід: крутний момент/швидкість занадто високі', class WarningCrane, trigger "AlarmsWord2" bit 7
   328: '4UZ2 (A07922) - Привід: крутний момент/швидкість поза межами допуску', class WarningCrane, trigger "AlarmsWord2" bit 8
   329: '4UZ2 (A07927) - DC гальмівний активний', class WarningCrane, trigger "AlarmsWord2" bit 9
   330: '4UZ2 (A07980) - Привід: Обертовий вимірювання активовано', class WarningCrane, trigger "AlarmsWord2" bit 10
   331: '4UZ2 (A07981) - Привід: Увімкнути сигнали для обертовий вимірювання відсутній', class WarningCrane, trigger "AlarmsWord2" bit 11
   332: '4UZ2 (A07991) - Привід: Ідентифікація даних двигуна активовано', class WarningCrane, trigger "AlarmsWord2" bit 12
   333: '4UZ2 (A08511) - PN/COMM BOARD: Приймання конфігурація дані некоректний', class WarningCrane, trigger "AlarmsWord2" bit 13
   334: '4UZ2 (A08526) - PN/COMM BOARD: Відсутній циклічний з’єднання', class WarningCrane, trigger "AlarmsWord2" bit 14
   335: '4UZ2 (A08565) - PNCOMM BOARD: Узгодженість помилка що впливає на регульований параметри', class WarningCrane, trigger "AlarmsWord2" bit 15
   336: '4UZ2 (A30049) - Силовий модуль: несправний внутрішній вентилятор', class WarningCrane, trigger "AlarmsWord3" bit 0
   337: '4UZ2 (A30502) - Силовий модуль: Перенапруга кола постійного струму', class WarningCrane, trigger "AlarmsWord3" bit 1
   338: '4UZ2 (A30920) - Силовий модуль: несправність датчика температури', class WarningCrane, trigger "AlarmsWord3" bit 2
   339: '4UZ2 (F01000) - Внутрішня програмна помилка', class ErrorCrane, trigger "FaultsWord1" bit 0
   340: '4UZ2 (F01001) - Виняток операції з плаваючою комою', class ErrorCrane, trigger "FaultsWord1" bit 1
   341: '4UZ2 (F01015) - Внутрішня програмна помилка', class ErrorCrane, trigger "FaultsWord1" bit 2
   342: '4UZ2 (F01033) - Перемикання одиниць: некоректне опорне значення параметра', class ErrorCrane, trigger "FaultsWord1" bit 3
   343: '4UZ2 (F01034) - Перемикання одиниць: не вдалося обчислити значення параметрів після зміни опорного значення', class ErrorCrane, trigger "FaultsWord1" bit 4
   344: '4UZ2 (F01040) - Збережіть налаштування параметрів і виконайте повторне увімкнення живлення', class ErrorCrane, trigger "FaultsWord1" bit 5
   345: '4UZ2 (F01044) - CU: Помилка описових даних', class ErrorCrane, trigger "FaultsWord1" bit 6
   346: '4UZ2 (F01054) - CU: Перевищено системне обмеження', class ErrorCrane, trigger "FaultsWord1" bit 7
   347: '4UZ2 (F01105) - CU: Недостатньо пам’яті', class ErrorCrane, trigger "FaultsWord1" bit 8
   348: '4UZ2 (F01122) - Частота на вході вимірювального щупа занадто висока', class ErrorCrane, trigger "FaultsWord1" bit 9
   349: '4UZ2 (F01205) - CU: Переповнення часового кванта', class ErrorCrane, trigger "FaultsWord1" bit 10
   350: '4UZ2 (F01250) - CU: Некоректні дані CU-EEPROM, доступні лише для читання', class ErrorCrane, trigger "FaultsWord1" bit 11
   351: '4UZ2 (F01512) - BICO: масштабування недоступне', class ErrorCrane, trigger "FaultsWord1" bit 12
   352: '4UZ2 (F01600) - SI P1 (CU): Ініційовано зупинку A', class ErrorCrane, trigger "FaultsWord1" bit 13
   353: '4UZ2 (F01625) - SI P1 (CU): Помилка сигналу справності в даних безпеки', class ErrorCrane, trigger "FaultsWord1" bit 14
   354: '4UZ2 (F01650) - SI P1 (CU): Потрібне приймальне випробування', class ErrorCrane, trigger "FaultsWord1" bit 15
   355: '4UZ2 (F01659) - SI P1 (CU): Запит на запис параметра відхилено', class ErrorCrane, trigger "FaultsWord2" bit 0
   356: '4UZ2 (F01666) - SI Motion P1 (CU): Постійний сигнал «1» на F-DI для безпечного квитування', class ErrorCrane, trigger "FaultsWord2" bit 1
   357: '4UZ2 (F01910) - Польова шина: тайм-аут заданого значення', class ErrorCrane, trigger "FaultsWord2" bit 2
   358: '4UZ2 (F01910) - Ввід: напругу живлення (p0210) параметризовано некоректно', class ErrorCrane, trigger "FaultsWord2" bit 3
   359: '4UZ2 (F07011) - Привід: перегрів двигуна', class ErrorCrane, trigger "FaultsWord2" bit 4
   360: '4UZ2 (F07016) - Привід: Несправність датчика температури двигуна', class ErrorCrane, trigger "FaultsWord2" bit 5
   361: '4UZ2 (F07086) - Перемикання одиниць: порушення обмеження параметра через зміну опорного значення', class ErrorCrane, trigger "FaultsWord2" bit 6
   362: '4UZ2 (F07088) - Перемикання одиниць: порушення обмеження параметра через перемикання одиниць', class ErrorCrane, trigger "FaultsWord2" bit 7
   363: '4UZ2 (F07320) - Привід: Автоматичний перезапуск перервано', class ErrorCrane, trigger "FaultsWord2" bit 8
   364: '4UZ2 (F07330) - Підхоплення обертового двигуна: виміряний пошуковий струм занадто малий', class ErrorCrane, trigger "FaultsWord2" bit 9
   365: '4UZ2 (F07426) - Технологія регулятор фактичний значення обмежений', class ErrorCrane, trigger "FaultsWord2" bit 10
   366: '4UZ2 (F07801) - Привід: Двигун Перевищення струму', class ErrorCrane, trigger "FaultsWord2" bit 11
   367: '4UZ2 (F07801) - Привід: виявлено коротке замикання/замикання на землю', class ErrorCrane, trigger "FaultsWord2" bit 12
   368: '4UZ2 (F07860) - Зовнішній несправність 1', class ErrorCrane, trigger "FaultsWord2" bit 13
   369: '4UZ2 (F07861) - Зовнішній несправність 2', class ErrorCrane, trigger "FaultsWord2" bit 14
   370: '4UZ2 (F07861) - Зовнішній несправність 3', class ErrorCrane, trigger "FaultsWord2" bit 15
   371: '4UZ2 (F07900) - Привід: заклинювання двигуна/регулятор швидкості на межі', class ErrorCrane, trigger "FaultsWord3" bit 0
   372: '4UZ2 (F07901) - Привід: перевищення швидкості двигуна', class ErrorCrane, trigger "FaultsWord3" bit 1
   373: '4UZ2 (F07902) - Привід: двигун зупинився', class ErrorCrane, trigger "FaultsWord3" bit 2
   374: '4UZ2 (F07923) - Привід: крутний момент/швидкість занадто низькі', class ErrorCrane, trigger "FaultsWord3" bit 3
   375: '4UZ2 (F07924) - Привід: крутний момент/швидкість занадто високі', class ErrorCrane, trigger "FaultsWord3" bit 4
   376: '4UZ2 (F08501) - PN/COMM BOARD: тайм-аут заданого значення', class ErrorCrane, trigger "FaultsWord3" bit 5
   377: '4UZ2 (F08502) - PN/COMM BOARD: закінчився контрольний час сигналу справності', class ErrorCrane, trigger "FaultsWord3" bit 6
   378: '4UZ2 (F06210) - Ввід: Сумування струм занадто високий', class ErrorCrane, trigger "FaultsWord3" bit 7
   379: '4UZ2 (F13100) - Захист ноу-хау: помилка захисту від копіювання', class ErrorCrane, trigger "FaultsWord3" bit 8
   380: '4UZ2 (F13101) - Захист ноу-хау: неможливо активувати захист від копіювання', class ErrorCrane, trigger "FaultsWord3" bit 9
   381: '4UZ2 (F30001) - Силовий модуль: перевищення струму', class ErrorCrane, trigger "FaultsWord3" bit 10
   382: '4UZ2 (F30002) - Силовий модуль: перенапруга кола постійного струму', class ErrorCrane, trigger "FaultsWord3" bit 11
   383: '4UZ2 (F30003) - Силовий модуль: занижена напруга кола постійного струму', class ErrorCrane, trigger "FaultsWord3" bit 12
   384: '4UZ2 (F30004) - Силовий модуль: перегрів радіатора інвертора AC', class ErrorCrane, trigger "FaultsWord3" bit 13
   385: '4UZ2 (F30005) - Силовий модуль: перевантаження I²t', class ErrorCrane, trigger "FaultsWord3" bit 14
   386: '4UZ2 (F30011) - Силовий модуль: відсутня фаза мережі в головному колі', class ErrorCrane, trigger "FaultsWord3" bit 15
   387: '4UZ2 (F30015) - Силовий модуль: відсутня фаза кабелю двигуна', class ErrorCrane, trigger "FaultsWord4" bit 0
   388: '4UZ2 (F30021) - Силовий модуль: замикання на землю', class ErrorCrane, trigger "FaultsWord4" bit 1
   389: '4UZ2 (F30022) - Силовий модуль: контроль Uce', class ErrorCrane, trigger "FaultsWord4" bit 2
   390: '4UZ2 (F30027) - Силовий модуль: контроль часу попереднього заряду кола постійного струму', class ErrorCrane, trigger "FaultsWord4" bit 3
   391: '4UZ2 (F30035) - Силовий модуль: перегрів повітря на вході', class ErrorCrane, trigger "FaultsWord4" bit 4
   392: '4UZ2 (F30036) - Силовий модуль: внутрішній перегрів', class ErrorCrane, trigger "FaultsWord4" bit 5
   393: '4UZ2 (F30037) - Силовий модуль: перегрів випрямляча', class ErrorCrane, trigger "FaultsWord4" bit 6
   394: '4UZ2 (F30052) - Помилка даних EEPROM', class ErrorCrane, trigger "FaultsWord4" bit 7
   395: '4UZ2 (F30053) - FPGA дані несправний', class ErrorCrane, trigger "FaultsWord4" bit 8
   396: '4UZ2 (F30059) - Силовий модуль: несправний внутрішній вентилятор', class ErrorCrane, trigger "FaultsWord4" bit 9
   397: '4UZ2 (F30074) - Помилка зв’язку між Керування Модуль та Силовий модуль', class ErrorCrane, trigger "FaultsWord4" bit 10
   398: '4UZ2 (F30600) - SI P2: Ініційовано зупинку A', class ErrorCrane, trigger "FaultsWord4" bit 11
   399: '4UZ2 (F30664) - Помилка під час завантаження', class ErrorCrane, trigger "FaultsWord4" bit 12
   400: '4UZ2 (F30850) - Силовий модуль: Внутрішня програмна помилка', class ErrorCrane, trigger "FaultsWord4" bit 13
   401: '4UZ2 (F06211) - Ввід: сумарний струм неприпустимо високий', class ErrorCrane, trigger "FaultsWord4" bit 14
   402: '4UZ2 (F08510) - PN/COMM BOARD: некоректні дані конфігурації передавання', class ErrorCrane, trigger "FaultsWord4" bit 15
   479: 'Автомат. вим. 6SF1. Змінено стан з вимкн. на увімкн.', class MessageContactor, trigger "HMI_DB_Messages_LinearContactor_wMessageWord1" bit 0
   496: 'Автомат. вим. 6SF1. Змінено стан з увімкн. на вимкн.', class MessageContactor, trigger "HMI_DB_Messages_LinearContactor_wMessageWord1" bit 1
   529: 'Контроль наявності напруги 6KV у нормі', class MessageContactor, trigger "HMI_DB_Messages_LinearContactor_wMessageWord1" bit 2
   530: 'Похибка контролю наявності напруги 6KV', class MessageContactor, trigger "HMI_DB_Messages_LinearContactor_wMessageWord1" bit 3
   531: 'Автомат. вим. 6SF5. Змінено стан з вимкн. на увімкн.', class MessageContactor, trigger "HMI_DB_Messages_LinearContactor_wMessageWord1" bit 4
   532: 'Автомат. вим. 6SF5. Змінено стан з увімкн. на вимкн.', class MessageContactor, trigger "HMI_DB_Messages_LinearContactor_wMessageWord1" bit 5
   533: 'Автомат. вим. 6QF2. Змінено стан з вимкн. на увімкн.', class MessageContactor, trigger "HMI_DB_Messages_LinearContactor_wMessageWord1" bit 6
   534: 'Автомат. вим. 6QF2. Змінено стан з увімкн. на вимкн.', class MessageContactor, trigger "HMI_DB_Messages_LinearContactor_wMessageWord1" bit 7
   535: 'Автомат. вим. 6QF3. Змінено стан з вимкн. на увімкн.', class MessageContactor, trigger "HMI_DB_Messages_LinearContactor_wMessageWord1" bit 8
   536: 'Автомат. вим. 6QF3. Змінено стан з увімкн. на вимкн.', class MessageContactor, trigger "HMI_DB_Messages_LinearContactor_wMessageWord1" bit 9
   537: 'Сейсмодатчик у нормі', class MessageContactor, trigger "HMI_DB_Messages_LinearContactor_wMessageWord1" bit 10
   538: 'Сейсмодатчик помилка', class MessageContactor, trigger "HMI_DB_Messages_LinearContactor_wMessageWord1" bit 11
   539: 'Автомат. вим. 6SF2. Змінено стан з вимкн. на увімкн.', class MessageContactor, trigger "HMI_DB_Messages_LinearContactor_wMessageWord1" bit 12
   540: 'Автомат. вим. 6SF2. Змінено стан з увімкн. на вимкн.', class MessageContactor, trigger "HMI_DB_Messages_LinearContactor_wMessageWord1" bit 13
   541: 'Автомат. вим. 6SF4. Змінено стан з вимкн. на увімкн.', class MessageContactor, trigger "HMI_DB_Messages_LinearContactor_wMessageWord1" bit 14
   542: 'Автомат. вим. 6SF4. Змінено стан з увімкн. на вимкн.', class MessageContactor, trigger "HMI_DB_Messages_LinearContactor_wMessageWord1" bit 15
   544: 'Автомат. вим. 9QF4. Змінено стан з вимкн. на увімкн.', class MessageContactor, trigger "HMI_DB_Messages_LinearContactor_wMessageWord2" bit 0
   545: 'Автомат. вим. 9QF4. Змінено стан з увімкн. на вимкн.', class MessageContactor, trigger "HMI_DB_Messages_LinearContactor_wMessageWord2" bit 1
   546: 'Підігрів шафи SU1. Змінено стан з вимкн. на увімкн.', class MessageContactor, trigger "HMI_DB_Messages_LinearContactor_wMessageWord2" bit 2
   547: 'Підігрів шафи SU1. Змінено стан з увімкн. на вимкн.', class MessageContactor, trigger "HMI_DB_Messages_LinearContactor_wMessageWord2" bit 3
   548: 'Автомат. вим. 1QF1. Змінено стан з вимкн. на увімкн.', class MessageContactor, trigger "HMI_DB_Messages_LinearContactor_wMessageWord2" bit 4
   549: 'Автомат. вим. 1QF1. Змінено стан з увімкн. на вимкн.', class MessageContactor, trigger "HMI_DB_Messages_LinearContactor_wMessageWord2" bit 5
   550: 'Автомат. вим. 1QF2. Змінено стан з вимкн. на увімкн.', class MessageContactor, trigger "HMI_DB_Messages_LinearContactor_wMessageWord2" bit 6
   551: 'Автомат. вим. 1QF2. Змінено стан з увімкн. на вимкн.', class MessageContactor, trigger "HMI_DB_Messages_LinearContactor_wMessageWord2" bit 7
   552: 'Автомат. вим. 4QF1. Змінено стан з вимкн. на увімкн.', class MessageContactor, trigger "HMI_DB_Messages_LinearContactor_wMessageWord2" bit 8
   553: 'Автомат. вим. 4QF1. Змінено стан з увімкн. на вимкн.', class MessageContactor, trigger "HMI_DB_Messages_LinearContactor_wMessageWord2" bit 9
   554: 'Зв'язок по Profinet у нормі.', class MessageContactor, trigger "HMI_DB_Messages_LinearContactor_wMessageWord2" bit 10
   555: 'Помилка зв'язку по Profinet.', class MessageContactor, trigger "HMI_DB_Messages_LinearContactor_wMessageWord2" bit 11
   556: 'Нульове блокування відсутнє.', class MessageContactor, trigger "HMI_DB_Messages_LinearContactor_wMessageWord2" bit 12
   557: 'Нульове блокування присутнє.', class MessageContactor, trigger "HMI_DB_Messages_LinearContactor_wMessageWord2" bit 13
   558: 'Дозвіл роботи 3M1 (РП роз'єднаний з приводом)', class MessageContactor, trigger "HMI_DB_Messages_LinearContactor_wMessageWord2" bit 14
   559: 'Заборона роботи 3M1 (РП з'єднаний з приводом)', class MessageContactor, trigger "HMI_DB_Messages_LinearContactor_wMessageWord2" bit 15
   561: 'Дозвіл роботи 4M1 (РП роз'єднаний з приводом)', class MessageContactor, trigger "HMI_DB_Messages_LinearContactor_wMessageWord3" bit 0
   562: 'Заборона роботи 4M1 (РП з'єднаний з приводом)', class MessageContactor, trigger "HMI_DB_Messages_LinearContactor_wMessageWord3" bit 1
   563: 'Дозвіл роботи 4M2 (РП роз'єднаний з приводом)', class MessageContactor, trigger "HMI_DB_Messages_LinearContactor_wMessageWord3" bit 2
   564: 'Заборона роботи 4M2 (РП з'єднаний з приводом)', class MessageContactor, trigger "HMI_DB_Messages_LinearContactor_wMessageWord3" bit 3
   565: 'Кінц. вимик. дозволу роботи рух вправо 4SQ22 у нормі', class MessageContactor, trigger "HMI_DB_Messages_LinearContactor_wMessageWord3" bit 4
   566: 'Спрацював кінц. вимик. дозволу роботи рух вправо 4SQ22', class MessageContactor, trigger "HMI_DB_Messages_LinearContactor_wMessageWord3" bit 5
   567: 'Кінц. вимик. дозволу роботи рух вліво 4SQ21 у нормі', class MessageContactor, trigger "HMI_DB_Messages_LinearContactor_wMessageWord3" bit 6
   568: 'Спрацював кінц. вимик. дозволу роботи рух вліво 4SQ21', class MessageContactor, trigger "HMI_DB_Messages_LinearContactor_wMessageWord3" bit 7
   569: 'Автомат. вим. 6QF4. Змінено стан з вимкн. на увімкн.', class MessageContactor, trigger "HMI_DB_Messages_LinearContactor_wMessageWord3" bit 8
   570: 'Автомат. вим. 6QF4. Змінено стан з увімкн. на вимкн.', class MessageContactor, trigger "HMI_DB_Messages_LinearContactor_wMessageWord3" bit 9
   571: 'Кінц. вимик. дозволу роботи рух вниз 1SQ1.4 у нормі', class MessageContactor, trigger "HMI_DB_Messages_LinearContactor_wMessageWord3" bit 10
   572: 'Спрацював кінц. вимик. дозволу роботи рух вниз 1SQ1.4', class MessageContactor, trigger "HMI_DB_Messages_LinearContactor_wMessageWord3" bit 11
   573: 'Кінц. вимик. дозволу роботи рух вгору 1SQ1.3 у нормі', class MessageContactor, trigger "HMI_DB_Messages_LinearContactor_wMessageWord3" bit 12
   574: 'Спрацював кінц. вимик. дозволу роботи рух вгору 1SQ1.3', class MessageContactor, trigger "HMI_DB_Messages_LinearContactor_wMessageWord3" bit 13
   575: 'Кінц. вимик. дозволу роботи рух назад 3SQ2.2 у нормі', class MessageContactor, trigger "HMI_DB_Messages_LinearContactor_wMessageWord3" bit 14
   576: 'Спрацював кінц. вимик. дозволу роботи рух назад 3SQ2.2', class MessageContactor, trigger "HMI_DB_Messages_LinearContactor_wMessageWord3" bit 15
   577: 'Кінц. вимик. дозволу роботи рух вперед 3SQ1.2 у нормі', class MessageContactor, trigger "HMI_DB_Messages_LinearContactor_wMessageWord4" bit 0
   578: 'Спрацював кінц. вимик. дозволу роботи рух вперед 3SQ1.2', class MessageContactor, trigger "HMI_DB_Messages_LinearContactor_wMessageWord4" bit 1
   579: 'Дозвіл роботи (МРР роз'єднаний з гальмом (1YB2))', class MessageContactor, trigger "HMI_DB_Messages_LinearContactor_wMessageWord4" bit 2
   580: 'Заборона роботи (МРР з'єднаний з гальмом (1YB2))', class MessageContactor, trigger "HMI_DB_Messages_LinearContactor_wMessageWord4" bit 3
   581: 'Дозвіл роботи механізму підйому (РП)', class MessageContactor, trigger "HMI_DB_Messages_LinearContactor_wMessageWord4" bit 4
   582: 'Заборона роботи механізму підйому (РП)', class MessageContactor, trigger "HMI_DB_Messages_LinearContactor_wMessageWord4" bit 5
   583: 'Таймаут увімкнення контактора 6KM1 або спрцювання кнопки 6SB3 / Таймаут увімкнення контактора 6KM1', class ErrorContactor, trigger "HMI_DB_Alarms_Contactor_AlarmWord1" bit 0
   600: 'Команда на увімкн. лінійного контактору 6КМ1', class MessageContactor, trigger "HMI_DB_Messages_LinearContactor_wMessageWord4" bit 6
   601: 'Команда на вимкн. лінійного контактору 6КМ1', class MessageContactor, trigger "HMI_DB_Messages_LinearContactor_wMessageWord4" bit 7
   584: 'Відсутній або зник сигнал контактора 6КМ2', class ErrorContactor, trigger "HMI_DB_Alarms_Contactor_AlarmWord1" bit 1
   585: 'Спрацював автомат. вим. 6SF1 - живлення 6KV', class ErrorContactor, trigger "HMI_DB_Alarms_Contactor_AlarmWord1" bit 2
   586: 'Спрацювало реле 6KV - вхідна напруга не в нормі / Спрацювало реле 6KV - контроль напруги введення', class ErrorContactor, trigger "HMI_DB_Alarms_Contactor_AlarmWord1" bit 3
   587: 'Спрацював автомат. вим. 6SF5 - живлення кіл обгіріву', class ErrorContactor, trigger "HMI_DB_Alarms_Contactor_AlarmWord1" bit 4
   588: 'Спрацював автомат. вим. 6QF2 - захист кіл гальм', class ErrorContactor, trigger "HMI_DB_Alarms_Contactor_AlarmWord1" bit 5
   589: 'Спрацював автомат. вим. 6QF3 - вимикач трансф. 6T1', class ErrorContactor, trigger "HMI_DB_Alarms_Contactor_AlarmWord1" bit 6
   590: 'Спрацював автомат. вим. 6QF4 - вимикач втор. кіл трансф. 6T1', class ErrorContactor, trigger "HMI_DB_Alarms_Contactor_AlarmWord1" bit 7
   591: 'Спрацював автомат. вим. 6SF2 - вимикач кіл управління 220в', class ErrorContactor, trigger "HMI_DB_Alarms_Contactor_AlarmWord1" bit 8
   592: 'Спрацював автомат. вим. 6SF4 - вимикач кіл живлення ОВП', class ErrorContactor, trigger "HMI_DB_Alarms_Contactor_AlarmWord1" bit 9
   593: 'Спрацював автомат. вим. 9QF4 - вимикач власн. потреб шафи', class ErrorContactor, trigger "HMI_DB_Alarms_Contactor_AlarmWord1" bit 10
   594: 'Спрацював автомат. вим. 1QF1 - захист випрямляча гальма 1YB1', class ErrorContactor, trigger "HMI_DB_Alarms_Contactor_AlarmWord1" bit 11
   595: 'Спрацював автомат. вим. 1QF2 - захист випрямляча гальма 1YB2', class ErrorContactor, trigger "HMI_DB_Alarms_Contactor_AlarmWord1" bit 12
   596: 'Спрацював автомат. вим. 4QF1 - захист кіл гальм', class ErrorContactor, trigger "HMI_DB_Alarms_Contactor_AlarmWord1" bit 13
   597: 'Спрацював кінц. вим. 1SQ33 - гальмо 1YB2 дозв. роб. (МРР роз'єд. з гальм)', class ErrorContactor, trigger "HMI_DB_Alarms_Contactor_AlarmWord1" bit 14
   598: 'Спрацював кінц. вим. 1SQ41 - дозвіл роботи мех. підйому, ручн. привід', class ErrorContactor, trigger "HMI_DB_Alarms_Contactor_AlarmWord1" bit 15
   604: 'Спрацював кінц. вим. 3SQ41 - дозвіл роботи мех. візка, ручн. привід', class ErrorContactor, trigger "HMI_DB_Alarms_Contactor_AlarmWord2" bit 0
   605: 'Спрацював кінц. вим. 4SQ41 - дозвіл роботи мех. крану, ручн. привід', class ErrorContactor, trigger "HMI_DB_Alarms_Contactor_AlarmWord2" bit 1
   606: 'Спрацював кінц. вим. 4SQ42 - дозвіл роботи мех. крану, ручн. привід', class ErrorContactor, trigger "HMI_DB_Alarms_Contactor_AlarmWord2" bit 2
   607: 'Спрацював кінц. вим. 1SQ13 - дозвіл роботи підйому, pух вгору', class ErrorContactor, trigger "HMI_DB_Alarms_Contactor_AlarmWord2" bit 3
   608: 'Спрацював кінц. вим. 1SQ14 - дозвіл роботи підйому, pух вниз', class ErrorContactor, trigger "HMI_DB_Alarms_Contactor_AlarmWord2" bit 4
   609: 'Спрацював кінц. вим. 3SQ12 - дозвіл роботи візка, рух вперед', class ErrorContactor, trigger "HMI_DB_Alarms_Contactor_AlarmWord2" bit 5
   610: 'Спрацював кінц. вим. 3SQ22 - дозвіл роботи візка, рух назад', class ErrorContactor, trigger "HMI_DB_Alarms_Contactor_AlarmWord2" bit 6
   611: 'Спрацював кінц. вим. 4SQ21 - дозвіл роботи моста, рух вліво', class ErrorContactor, trigger "HMI_DB_Alarms_Contactor_AlarmWord2" bit 7
   612: 'Спрацював кінц. вим. 4SQ22 - дозвіл роботи моста, рух вправо', class ErrorContactor, trigger "HMI_DB_Alarms_Contactor_AlarmWord2" bit 8
   613: 'Спрацював сейсмодатчик', class ErrorContactor, trigger "HMI_DB_Alarms_Contactor_AlarmWord2" bit 9
   614: 'Критична помилка або втрата зв'язку Profinet', class ErrorContactor, trigger "HMI_DB_Alarms_Contactor_AlarmWord2" bit 10
   413: 'Лінійний контактор 6КМ1. Змінено стан з вимкн. на увімкн.', class MessageContactor, trigger "HMI_DB_Messages_LinearContactor_wMessageWord4" bit 8
   430: 'Лінійний контактор 6КМ1. Змінено стан з увімкн. на вимкн.', class MessageContactor, trigger "HMI_DB_Messages_LinearContactor_wMessageWord4" bit 9
   447: 'Лінійний контактор 6КМ2. Змінено стан з вимкн. на увімкн.', class MessageContactor, trigger "HMI_DB_Messages_LinearContactor_wMessageWord4" bit 10
   464: 'Лінійний контактор 6КМ2. Змінено стан з увімкн. на вимкн.', class MessageContactor, trigger "HMI_DB_Messages_LinearContactor_wMessageWord4" bit 11
   543: 'Команда "Підйом" подана', class MessageLiftUp, trigger "HMI_DB_Messages_LiftUp_wMessageWord1" bit 0
   560: 'Команда "Підйом" знята', class MessageLiftUp, trigger "HMI_DB_Messages_LiftUp_wMessageWord1" bit 1
   599: 'Команда "Спуск" подана', class MessageLiftUp, trigger "HMI_DB_Messages_LiftUp_wMessageWord1" bit 2
   602: 'Команда "Спуск" знята', class MessageLiftUp, trigger "HMI_DB_Messages_LiftUp_wMessageWord1" bit 3
   603: 'Команда "Підйом" 2-га швидкість подана', class MessageLiftUp, trigger "HMI_DB_Messages_LiftUp_wMessageWord1" bit 4
   615: 'Команда "Підйом" 2-га швидкість знята', class MessageLiftUp, trigger "HMI_DB_Messages_LiftUp_wMessageWord1" bit 5
   616: 'Команда "Спуск" 2-га швидкість подана', class MessageLiftUp, trigger "HMI_DB_Messages_LiftUp_wMessageWord1" bit 6
   617: 'Команда "Спуск" 2-га швидкість знята', class MessageLiftUp, trigger "HMI_DB_Messages_LiftUp_wMessageWord1" bit 7
   618: 'Спрацював термозахист гальм. резистора 1BT1', class MessageLiftUp, trigger "HMI_DB_Messages_LiftUp_wMessageWord1" bit 8
   619: 'Термозахист гальм. резистора 1BT1 у нормі', class MessageLiftUp, trigger "HMI_DB_Messages_LiftUp_wMessageWord1" bit 9
   620: 'Термозахист двигуна 1M1 у нормі', class MessageLiftUp, trigger "HMI_DB_Messages_LiftUp_wMessageWord1" bit 10
   621: 'Спрацював термозахист двигуна 1M1', class MessageLiftUp, trigger "HMI_DB_Messages_LiftUp_wMessageWord1" bit 11
   622: 'Кінц. вимик. товщин. гальм. накладок 1SQ23 у нормі', class MessageLiftUp, trigger "HMI_DB_Messages_LiftUp_wMessageWord1" bit 12
   623: 'Спрацював кінц. вимик. товщин. гальм. накладок 1SQ23', class MessageLiftUp, trigger "HMI_DB_Messages_LiftUp_wMessageWord1" bit 13
   624: 'Робоче гальмо розагальмоване', class MessageLiftUp, trigger "HMI_DB_Messages_LiftUp_wMessageWord1" bit 14
   625: 'Робоче гальмо загальмоване', class MessageLiftUp, trigger "HMI_DB_Messages_LiftUp_wMessageWord1" bit 15
   628: 'Ослабення канатів 1К12 у нормі.', class MessageLiftUp, trigger "HMI_DB_Messages_LiftUp_wMessageWord2" bit 0
   629: 'Спрацював датчик послаблення канатів 1К12', class MessageLiftUp, trigger "HMI_DB_Messages_LiftUp_wMessageWord2" bit 1
   630: 'Перевищення вантажу 1К11 у нормі', class MessageLiftUp, trigger "HMI_DB_Messages_LiftUp_wMessageWord2" bit 2
   631: 'Спрацювало перевищення кантажу 1К11', class MessageLiftUp, trigger "HMI_DB_Messages_LiftUp_wMessageWord2" bit 3
   632: 'Калібровка мех. підйому у нормі.', class MessageLiftUp, trigger "HMI_DB_Messages_LiftUp_wMessageWord2" bit 4
   633: 'Мех. підйому втратив калібровку', class MessageLiftUp, trigger "HMI_DB_Messages_LiftUp_wMessageWord2" bit 5
   634: 'Помилка ПЧ підйому 1UZ1', class MessageLiftUp, trigger "HMI_DB_Messages_LiftUp_wMessageWord2" bit 6
   635: 'ПЧ підйому 1UZ1 працює без помилок', class MessageLiftUp, trigger "HMI_DB_Messages_LiftUp_wMessageWord2" bit 7
   636: 'Кінц. вимик. дозвіл ном. швидк. рух угору 1SQ1.1 у нормі', class MessageLiftUp, trigger "HMI_DB_Messages_LiftUp_wMessageWord2" bit 8
   637: 'Спрацював кінц. вимик. дозвіл ном. швидк. рух угору 1SQ1.1', class MessageLiftUp, trigger "HMI_DB_Messages_LiftUp_wMessageWord2" bit 9
   638: 'Кінц. вимик. дозвіл ном. швидк. рух вниз 1SQ1.2 у нормі', class MessageLiftUp, trigger "HMI_DB_Messages_LiftUp_wMessageWord2" bit 10
   639: 'Спрацював кінц. вимик. дозвіл ном. швидк. рух вниз 1SQ1.2', class MessageLiftUp, trigger "HMI_DB_Messages_LiftUp_wMessageWord2" bit 11
   640: 'Кінц. вимик. гальм розгальмоване 1SQ21 у нормі', class MessageLiftUp, trigger "HMI_DB_Messages_LiftUp_wMessageWord2" bit 12
   641: 'Спрацював кінц. вимик. гальм не розгальмоване 1SQ21', class MessageLiftUp, trigger "HMI_DB_Messages_LiftUp_wMessageWord2" bit 13
   642: 'Кінц. вимик. гальм загальмоване 1SQ22 у нормі', class MessageLiftUp, trigger "HMI_DB_Messages_LiftUp_wMessageWord2" bit 14
   643: 'Спрацював кінц. вимик. гальм не загальмоване 1SQ22', class MessageLiftUp, trigger "HMI_DB_Messages_LiftUp_wMessageWord2" bit 15
   645: 'Кінц. вимик. гальм розгальмоване 1SQ31 у нормі', class MessageLiftUp, trigger "HMI_DB_Messages_LiftUp_wMessageWord3" bit 0
   646: 'Спрацював кінц. вимик. гальм не розгальмоване 1SQ31', class MessageLiftUp, trigger "HMI_DB_Messages_LiftUp_wMessageWord3" bit 1
   647: 'Кінц. вимик. гальм загальмоване 1SQ32 у нормі', class MessageLiftUp, trigger "HMI_DB_Messages_LiftUp_wMessageWord3" bit 2
   648: 'Спрацював кінц. вимик. гальм не загальмоване 1SQ32', class MessageLiftUp, trigger "HMI_DB_Messages_LiftUp_wMessageWord3" bit 3
   626: '1UZ1 (A06205) - Ввід: провал напруги щонайменше в одній фазі мережі', class WarningLiftUp, trigger "AlarmsWord3" bit 3
   627: '1UZ1 (A06206) - Ввід: аварійне повідомлення про асиметрію струмів мережі', class WarningLiftUp, trigger "AlarmsWord3" bit 4
   644: '1UZ1 (A06208) - Ввід: аварійне повідомлення про асиметрію струмів мережі', class WarningLiftUp, trigger "AlarmsWord3" bit 5
   649: '1UZ1 (A06215) - Ввід: Сумування струм занадто високий', class WarningLiftUp, trigger "AlarmsWord3" bit 6
   650: '1UZ1 (A06250) - Ввід: несправний(і) конденсатор(и) щонайменше в одній фазі мережевого фільтра', class WarningLiftUp, trigger "AlarmsWord3" bit 7
   651: '1UZ1 (A06260) - Ввід: Температура у мережа фільтр занадто високий', class WarningLiftUp, trigger "AlarmsWord3" bit 8
   652: '1UZ1 (A06301) - Ввід: перенапруга мережі', class WarningLiftUp, trigger "AlarmsWord3" bit 9
   653: '1UZ1 (A06350) - Ввід: Виміряний Частота мережі занадто висока', class WarningLiftUp, trigger "AlarmsWord3" bit 10
   654: '1UZ1 (A06351) - Ввід: Виміряний Частота мережі занадто низька', class WarningLiftUp, trigger "AlarmsWord3" bit 11
   655: '1UZ1 (A06800) - Ввід: напруга кола постійного струму опустилася нижче порога аварійного повідомлення', class WarningLiftUp, trigger "AlarmsWord3" bit 12
   656: '1UZ1 (A30034) - Силовий модуль: внутрішній перегрів', class WarningLiftUp, trigger "AlarmsWord3" bit 13
   657: '1UZ1 (A30041) - Силовий модуль: аварійне повідомлення про занижену напругу 24 В', class WarningLiftUp, trigger "AlarmsWord3" bit 14
   658: '1UZ1 (A30042) - Силовий модуль: вентилятор досяг максимального напрацювання', class WarningLiftUp, trigger "AlarmsWord3" bit 15
   660: '1UZ1 (A30044) - Силовий модуль: аварійне повідомлення про перенапругу 24 В', class WarningLiftUp, trigger "AlarmsWord4" bit 0
   661: '1UZ1 (A30046) - Силовий модуль: аварійне повідомлення про занижену напругу', class WarningLiftUp, trigger "AlarmsWord4" bit 1
   662: '1UZ1 (A30077) - Силовий модуль: теплове перевантаження внутрішнього гальмівного резистора', class WarningLiftUp, trigger "AlarmsWord4" bit 2
   663: '1UZ1 (A30079) - Силовий модуль: відносно напруги живлення напруга кола постійного струму занадто висока', class WarningLiftUp, trigger "AlarmsWord4" bit 3
   664: '3UZ1 (A06205) - Ввід: провал напруги щонайменше в одній фазі мережі', class WarningTrolley, trigger "AlarmsWord3" bit 3
   665: '3UZ1 (A06206) - Ввід: аварійне повідомлення про асиметрію струмів мережі', class WarningTrolley, trigger "AlarmsWord3" bit 4
   666: '3UZ1 (A06208) - Ввід: аварійне повідомлення про асиметрію струмів мережі', class WarningTrolley, trigger "AlarmsWord3" bit 5
   667: '3UZ1 (A06215) - Ввід: Сумування струм занадто високий', class WarningTrolley, trigger "AlarmsWord3" bit 6
   668: '3UZ1 (A06250) - Ввід: несправний(і) конденсатор(и) щонайменше в одній фазі мережевого фільтра', class WarningTrolley, trigger "AlarmsWord3" bit 7
   669: '3UZ1 (A06260) - Ввід: Температура у мережа фільтр занадто високий', class WarningTrolley, trigger "AlarmsWord3" bit 8
   670: '3UZ1 (A06301) - Ввід: перенапруга мережі', class WarningTrolley, trigger "AlarmsWord3" bit 9
   671: '3UZ1 (A06350) - Ввід: Виміряний Частота мережі занадто висока', class WarningTrolley, trigger "AlarmsWord3" bit 10
   672: '3UZ1 (A06351) - Ввід: Виміряний Частота мережі занадто низька', class WarningTrolley, trigger "AlarmsWord3" bit 11
   673: '3UZ1 (A06800) - Ввід: напруга кола постійного струму опустилася нижче порога аварійного повідомлення', class WarningTrolley, trigger "AlarmsWord3" bit 12
   674: '3UZ1 (A30034) - Силовий модуль: внутрішній перегрів', class WarningTrolley, trigger "AlarmsWord3" bit 13
   675: '3UZ1 (A30041) - Силовий модуль: аварійне повідомлення про занижену напругу 24 В', class WarningTrolley, trigger "AlarmsWord3" bit 14
   676: '3UZ1 (A30042) - Силовий модуль: вентилятор досяг максимального напрацювання', class WarningTrolley, trigger "AlarmsWord3" bit 15
   677: '3UZ1 (A30044) - Силовий модуль: аварійне повідомлення про перенапругу 24 В', class WarningTrolley, trigger "AlarmsWord4" bit 0
   678: '3UZ1 (A30046) - Силовий модуль: аварійне повідомлення про занижену напругу', class WarningTrolley, trigger "AlarmsWord4" bit 1
   679: '3UZ1 (A30077) - Силовий модуль: теплове перевантаження внутрішнього гальмівного резистора', class WarningTrolley, trigger "AlarmsWord4" bit 2
   680: '3UZ1 (A30079) - Силовий модуль: відносно напруги живлення напруга кола постійного струму занадто висока', class WarningTrolley, trigger "AlarmsWord4" bit 3
   681: '4UZ1 (A06205) - Ввід: провал напруги щонайменше в одній фазі мережі', class WarningCrane, trigger "AlarmsWord3" bit 3
   682: '4UZ1 (A06206) - Ввід: аварійне повідомлення про асиметрію струмів мережі', class WarningCrane, trigger "AlarmsWord3" bit 4
   683: '4UZ1 (A06208) - Ввід: аварійне повідомлення про асиметрію струмів мережі', class WarningCrane, trigger "AlarmsWord3" bit 5
   684: '4UZ1 (A06215) - Ввід: Сумування струм занадто високий', class WarningCrane, trigger "AlarmsWord3" bit 6
   685: '4UZ1 (A06250) - Ввід: несправний(і) конденсатор(и) щонайменше в одній фазі мережевого фільтра', class WarningCrane, trigger "AlarmsWord3" bit 7
   686: '4UZ1 (A06260) - Ввід: Температура у мережа фільтр занадто високий', class WarningCrane, trigger "AlarmsWord3" bit 8
   687: '4UZ1 (A06301) - Ввід: перенапруга мережі', class WarningCrane, trigger "AlarmsWord3" bit 9
   688: '4UZ1 (A06350) - Ввід: Виміряний Частота мережі занадто висока', class WarningCrane, trigger "AlarmsWord3" bit 10
   689: '4UZ1 (A06351) - Ввід: Виміряний Частота мережі занадто низька', class WarningCrane, trigger "AlarmsWord3" bit 11
   690: '4UZ1 (A06800) - Ввід: напруга кола постійного струму опустилася нижче порога аварійного повідомлення', class WarningCrane, trigger "AlarmsWord3" bit 12
   691: '4UZ1 (A30034) - Силовий модуль: внутрішній перегрів', class WarningCrane, trigger "AlarmsWord3" bit 13
   692: '4UZ1 (A30041) - Силовий модуль: аварійне повідомлення про занижену напругу 24 В', class WarningCrane, trigger "AlarmsWord3" bit 14
   693: '4UZ1 (A30042) - Силовий модуль: вентилятор досяг максимального напрацювання', class WarningCrane, trigger "AlarmsWord3" bit 15
   694: '4UZ1 (A30044) - Силовий модуль: аварійне повідомлення про перенапругу 24 В', class WarningCrane, trigger "AlarmsWord4" bit 0
   695: '4UZ1 (A30046) - Силовий модуль: аварійне повідомлення про занижену напругу', class WarningCrane, trigger "AlarmsWord4" bit 1
   696: '4UZ1 (A30077) - Силовий модуль: теплове перевантаження внутрішнього гальмівного резистора', class WarningCrane, trigger "AlarmsWord4" bit 2
   697: '4UZ1 (A30079) - Силовий модуль: відносно напруги живлення напруга кола постійного струму занадто висока', class WarningCrane, trigger "AlarmsWord4" bit 3
   698: '4UZ2 (A06205) - Ввід: провал напруги щонайменше в одній фазі мережі', class WarningCrane, trigger "AlarmsWord3" bit 3
   699: '4UZ2 (A06206) - Ввід: аварійне повідомлення про асиметрію струмів мережі', class WarningCrane, trigger "AlarmsWord3" bit 4
   700: '4UZ2 (A06208) - Ввід: аварійне повідомлення про асиметрію струмів мережі', class WarningCrane, trigger "AlarmsWord3" bit 5
   701: '4UZ2 (A06215) - Ввід: Сумування струм занадто високий', class WarningCrane, trigger "AlarmsWord3" bit 6
   702: '4UZ2 (A06250) - Ввід: несправний(і) конденсатор(и) щонайменше в одній фазі мережевого фільтра', class WarningCrane, trigger "AlarmsWord3" bit 7
   703: '4UZ2 (A06260) - Ввід: Температура у мережа фільтр занадто високий', class WarningCrane, trigger "AlarmsWord3" bit 8
   704: '4UZ2 (A06301) - Ввід: перенапруга мережі', class WarningCrane, trigger "AlarmsWord3" bit 9
   705: '4UZ2 (A06350) - Ввід: Виміряний Частота мережі занадто висока', class WarningCrane, trigger "AlarmsWord3" bit 10
   706: '4UZ2 (A06351) - Ввід: Виміряний Частота мережі занадто низька', class WarningCrane, trigger "AlarmsWord3" bit 11
   707: '4UZ2 (A06800) - Ввід: напруга кола постійного струму опустилася нижче порога аварійного повідомлення', class WarningCrane, trigger "AlarmsWord3" bit 12
   708: '4UZ2 (A30034) - Силовий модуль: внутрішній перегрів', class WarningCrane, trigger "AlarmsWord3" bit 13
   709: '4UZ2 (A30041) - Силовий модуль: аварійне повідомлення про занижену напругу 24 В', class WarningCrane, trigger "AlarmsWord3" bit 14
   710: '4UZ2 (A30042) - Силовий модуль: вентилятор досяг максимального напрацювання', class WarningCrane, trigger "AlarmsWord3" bit 15
   711: '4UZ2 (A30044) - Силовий модуль: аварійне повідомлення про перенапругу 24 В', class WarningCrane, trigger "AlarmsWord4" bit 0
   712: '14UZ2 (A30046) - Силовий модуль: аварійне повідомлення про занижену напругу', class WarningCrane, trigger "AlarmsWord4" bit 1
   713: '4UZ2 (A30077) - Силовий модуль: теплове перевантаження внутрішнього гальмівного резистора', class WarningCrane, trigger "AlarmsWord4" bit 2
   714: '4UZ2 (A30079) - Силовий модуль: відносно напруги живлення напруга кола постійного струму занадто висока', class WarningCrane, trigger "AlarmsWord4" bit 3
   659: 'Аварійний стоп', class ErrorLiftUp, trigger "HMI_DB_Alarms_LiftUp_AlarmWord1" bit 0
   715: 'Головний контактор вимкнений під час роботи', class ErrorLiftUp, trigger "HMI_DB_Alarms_LiftUp_AlarmWord1" bit 1
   716: 'Перегрів гальмівного резистора підйому 1BT1', class ErrorLiftUp, trigger "HMI_DB_Alarms_LiftUp_AlarmWord1" bit 2
   717: 'Перегрів двигуна підйому 1M1 (1KT)', class ErrorLiftUp, trigger "HMI_DB_Alarms_LiftUp_AlarmWord1" bit 3
   718: 'Знос колодок робочого гальма (1SQ23)', class ErrorLiftUp, trigger "HMI_DB_Alarms_LiftUp_AlarmWord1" bit 4
   719: 'Знос вбудованого гальма двигуна (1BM1_6k)', class ErrorLiftUp, trigger "HMI_DB_Alarms_LiftUp_AlarmWord1" bit 5
   720: 'Контроль обертання барабану (1BV)', class ErrorLiftUp, trigger "HMI_DB_Alarms_LiftUp_AlarmWord1" bit 6
   721: 'Розбіжність датчика моменту 1А1 та ЧП > 20%', class ErrorLiftUp, trigger "HMI_DB_Alarms_LiftUp_AlarmWord1" bit 7
   722: 'Перевищення часу розгальмування робочого гальма', class ErrorLiftUp, trigger "HMI_DB_Alarms_LiftUp_AlarmWord1" bit 8
   723: 'Сигнал зносу гальм мех. підйому у нормі', class MessageLiftUp, trigger "HMI_DB_Messages_LiftUp_wMessageWord3" bit 4
   724: 'Сппрацював сигнал зносу гальма', class MessageLiftUp, trigger "HMI_DB_Messages_LiftUp_wMessageWord3" bit 5
   725: 'Сигнал контролю обертання барабану у нормі', class MessageLiftUp, trigger "HMI_DB_Messages_LiftUp_wMessageWord3" bit 6
   726: 'Спрацював сигнал контролю обертання барабану', class MessageLiftUp, trigger "HMI_DB_Messages_LiftUp_wMessageWord3" bit 7
   727: 'Механізм підйому почав рух з точки мм', class MessageLiftUp, trigger "HMI_DB_Messages_LiftUp_wMessageWord3" bit 8
   728: 'Механізм підйому закінчив рух у точці мм', class MessageLiftUp, trigger "HMI_DB_Messages_LiftUp_wMessageWord3" bit 9
   729: 'Активація рехимі калібровки для мех. підйому', class MessageLiftUp, trigger "HMI_DB_Messages_LiftUp_wMessageWord3" bit 10
   730: 'Деактивація рехимі калібровки для мех. підйому', class MessageLiftUp, trigger "HMI_DB_Messages_LiftUp_wMessageWord3" bit 11
   731: 'Помилка енкодеру підйому 1BR', class MessageLiftUp, trigger "HMI_DB_Messages_LiftUp_wMessageWord3" bit 12
   732: 'Енкодер підйому 1BR працює без помилок', class MessageLiftUp, trigger "HMI_DB_Messages_LiftUp_wMessageWord3" bit 13
   733: 'Не визначена позиція аварійних гальм', class ErrorLiftUp, trigger "HMI_DB_Alarms_LiftUp_AlarmWord1" bit 11
   734: 'Команда "Вперед" подана', class MessageTrolley, trigger "HMI_DB_Messages_Trolley_wMessageWord1" bit 0
   735: 'Команда "Вперед" знята', class MessageTrolley, trigger "HMI_DB_Messages_Trolley_wMessageWord1" bit 1
   736: 'Команда "Назад" подана', class MessageTrolley, trigger "HMI_DB_Messages_Trolley_wMessageWord1" bit 2
   737: 'Команда "Назад" знята', class MessageTrolley, trigger "HMI_DB_Messages_Trolley_wMessageWord1" bit 3
   738: 'Команда "Вперед" 2-га швидкість подана', class MessageTrolley, trigger "HMI_DB_Messages_Trolley_wMessageWord1" bit 4
   739: 'Команда "Вперед" 2-га швидкість знята', class MessageTrolley, trigger "HMI_DB_Messages_Trolley_wMessageWord1" bit 5
   740: 'Команда "Назад" 2-га швидкість подана', class MessageTrolley, trigger "HMI_DB_Messages_Trolley_wMessageWord1" bit 6
   741: 'Команда "Назад" 2-га швидкість знята', class MessageTrolley, trigger "HMI_DB_Messages_Trolley_wMessageWord1" bit 7
   742: 'Спрацював термозахист гальм. резистора 3BT1', class MessageTrolley, trigger "HMI_DB_Messages_Trolley_wMessageWord1" bit 8
   743: 'Термозахист гальм. резистора 3BT1 у нормі', class MessageTrolley, trigger "HMI_DB_Messages_Trolley_wMessageWord1" bit 9
   744: 'Термозахист двигуна 3M1 у нормі', class MessageTrolley, trigger "HMI_DB_Messages_Trolley_wMessageWord1" bit 10
   745: 'Спрацював термозахист двигуна 3M1', class MessageTrolley, trigger "HMI_DB_Messages_Trolley_wMessageWord1" bit 11
   746: 'Калібровка мех. візка у нормі.', class MessageTrolley, trigger "HMI_DB_Messages_Trolley_wMessageWord1" bit 12
   747: 'Мех. візка втратив калібровку', class MessageTrolley, trigger "HMI_DB_Messages_Trolley_wMessageWord1" bit 13
   748: 'Помилка ПЧ візка 3UZ1', class MessageTrolley, trigger "HMI_DB_Messages_Trolley_wMessageWord1" bit 14
   749: 'ПЧ візка 3UZ1 працює без помилок', class MessageTrolley, trigger "HMI_DB_Messages_Trolley_wMessageWord1" bit 15
   751: 'Кінц. вимик. дозвіл ном. швидк. рух вперед 3SQ1.1 у нормі', class MessageTrolley, trigger "HMI_DB_Messages_Trolley_wMessageWord2" bit 0
   752: 'Спрацював кінц. вимик. дозвіл ном. швидк. рух вперед 3SQ1.1', class MessageTrolley, trigger "HMI_DB_Messages_Trolley_wMessageWord2" bit 1
   753: 'Кінц. вимик. дозвіл ном. швидк. рух назад 3SQ2.1 у нормі', class MessageTrolley, trigger "HMI_DB_Messages_Trolley_wMessageWord2" bit 2
   754: 'Спрацював кінц. вимик. дозвіл ном. швидк. рух назад 3SQ2.1', class MessageTrolley, trigger "HMI_DB_Messages_Trolley_wMessageWord2" bit 3
   755: 'Механізм візка почав рух з точки мм', class MessageTrolley, trigger "HMI_DB_Messages_Trolley_wMessageWord2" bit 4
   756: 'Механізм візка закінчив рух у точці мм', class MessageTrolley, trigger "HMI_DB_Messages_Trolley_wMessageWord2" bit 5
   757: 'Активація рехимі калібровки для мех. візка', class MessageTrolley, trigger "HMI_DB_Messages_Trolley_wMessageWord2" bit 6
   758: 'Деактивація рехимі калібровки для мех. візка', class MessageTrolley, trigger "HMI_DB_Messages_Trolley_wMessageWord2" bit 7
   759: 'Помилка енкодеру візка 3BR', class MessageTrolley, trigger "HMI_DB_Messages_Trolley_wMessageWord2" bit 8
   760: 'Енкодер візка 3BR працює без помилок', class MessageTrolley, trigger "HMI_DB_Messages_Trolley_wMessageWord2" bit 9
   761: 'Несправність частотного перетворювача 1UZ1', class ErrorLiftUp, trigger "HMI_DB_Alarms_LiftUp_AlarmWord1" bit 9
   762: 'Несправність енкодера 1BR / Несправність енкодера BR1', class ErrorLiftUp, trigger "HMI_DB_Alarms_LiftUp_AlarmWord1" bit 10
   750: 'Аварійний стоп', class ErrorTrolley, trigger "HMI_DB_Alarms_Trolley_AlarmWord1" bit 0
   763: 'Головний контактор вимкнений під час роботи', class ErrorTrolley, trigger "HMI_DB_Alarms_Trolley_AlarmWord1" bit 1
   764: 'Перегрів гальмівного резистора візка 3BT1', class ErrorTrolley, trigger "HMI_DB_Alarms_Trolley_AlarmWord1" bit 2
   765: 'Перегрів двигуна візка 3M1 (3KT)', class ErrorTrolley, trigger "HMI_DB_Alarms_Trolley_AlarmWord1" bit 3
   766: 'Несправність частотного перетворювача 3UZ1', class ErrorTrolley, trigger "HMI_DB_Alarms_Trolley_AlarmWord1" bit 4
   767: 'Несправність енкодера 3BR', class ErrorTrolley, trigger "HMI_DB_Alarms_Trolley_AlarmWord1" bit 5
   768: 'Команда "Вліво" подана', class MessageCrane, trigger "HMI_DB_Messages_Crane_wMessageWord1" bit 0
   769: 'Команда "Вліво" знята', class MessageCrane, trigger "HMI_DB_Messages_Crane_wMessageWord1" bit 1
   770: 'Команда "Вправо" подана', class MessageCrane, trigger "HMI_DB_Messages_Crane_wMessageWord1" bit 2
   771: 'Команда "Вправо" знята', class MessageCrane, trigger "HMI_DB_Messages_Crane_wMessageWord1" bit 3
   772: 'Команда "Вліво" 2-га швидкість подана', class MessageCrane, trigger "HMI_DB_Messages_Crane_wMessageWord1" bit 4
   773: 'Команда "Вліво" 2-га швидкість знята', class MessageCrane, trigger "HMI_DB_Messages_Crane_wMessageWord1" bit 5
   774: 'Команда "Вправо" 2-га швидкість подана', class MessageCrane, trigger "HMI_DB_Messages_Crane_wMessageWord1" bit 6
   775: 'Команда "Вправо" 2-га швидкість знята', class MessageCrane, trigger "HMI_DB_Messages_Crane_wMessageWord1" bit 7
   776: 'Спрацював термозахист гальм. резистора 4BT1', class MessageCrane, trigger "HMI_DB_Messages_Crane_wMessageWord1" bit 8
   777: 'Термозахист гальм. резистора 4BT1 у нормі', class MessageCrane, trigger "HMI_DB_Messages_Crane_wMessageWord1" bit 9
   778: 'Спрацював термозахист гальм. резистора 4BT2', class MessageCrane, trigger "HMI_DB_Messages_Crane_wMessageWord1" bit 10
   779: 'Термозахист гальм. резистора 4BT2 у нормі', class MessageCrane, trigger "HMI_DB_Messages_Crane_wMessageWord1" bit 11
   780: 'Термозахист двигуна 4M1 у нормі', class MessageCrane, trigger "HMI_DB_Messages_Crane_wMessageWord1" bit 12
   781: 'Спрацював термозахист двигуна 4M1', class MessageCrane, trigger "HMI_DB_Messages_Crane_wMessageWord1" bit 13
   782: 'Термозахист двигуна 4M2 у нормі', class MessageCrane, trigger "HMI_DB_Messages_Crane_wMessageWord1" bit 14
   783: 'Спрацював термозахист двигуна 4M2', class MessageCrane, trigger "HMI_DB_Messages_Crane_wMessageWord1" bit 15
   786: 'Калібровка мех. крану у нормі.', class MessageCrane, trigger "HMI_DB_Messages_Crane_wMessageWord2" bit 0
   787: 'Мех. крану втратив калібровку', class MessageCrane, trigger "HMI_DB_Messages_Crane_wMessageWord2" bit 1
   788: 'Помилка ПЧ візка 4UZ1', class MessageCrane, trigger "HMI_DB_Messages_Crane_wMessageWord2" bit 2
   789: 'ПЧ візка 4UZ1 працює без помилок', class MessageCrane, trigger "HMI_DB_Messages_Crane_wMessageWord2" bit 3
   790: 'Помилка ПЧ візка 4UZ2', class MessageCrane, trigger "HMI_DB_Messages_Crane_wMessageWord2" bit 4
   791: 'ПЧ візка 4UZ2 працює без помилок', class MessageCrane, trigger "HMI_DB_Messages_Crane_wMessageWord2" bit 5
   792: 'Кінц. вимик. дозвіл ном. швидк. рух вліво 4SQ1.1 у нормі', class MessageCrane, trigger "HMI_DB_Messages_Crane_wMessageWord2" bit 6
   793: 'Спрацював кінц. вимик. дозвіл ном. швидк. рух вліво 4SQ1.1', class MessageCrane, trigger "HMI_DB_Messages_Crane_wMessageWord2" bit 7
   794: 'Кінц. вимик. дозвіл ном. швидк. рух вправо 4SQ1.2 у нормі', class MessageCrane, trigger "HMI_DB_Messages_Crane_wMessageWord2" bit 8
   795: 'Спрацював кінц. вимик. дозвіл ном. швидк. рух вправо 4SQ1.2', class MessageCrane, trigger "HMI_DB_Messages_Crane_wMessageWord2" bit 9
   796: 'Механізм крану почав рух з точки мм (4BR1)', class MessageCrane, trigger "HMI_DB_Messages_Crane_wMessageWord2" bit 10
   797: 'Механізм крану закінчив рух у точці мм (4BR1)', class MessageCrane, trigger "HMI_DB_Messages_Crane_wMessageWord2" bit 11
   798: 'Механізм крану почав рух з точки мм (4BR2)', class MessageCrane, trigger "HMI_DB_Messages_Crane_wMessageWord2" bit 12
   799: 'Механізм крану закінчив рух у точці мм (4BR2)', class MessageCrane, trigger "HMI_DB_Messages_Crane_wMessageWord2" bit 13
   800: 'Активація рехимі калібровки для мех. крану', class MessageCrane, trigger "HMI_DB_Messages_Crane_wMessageWord2" bit 14
   801: 'Деактивація рехимі калібровки для мех. крану', class MessageCrane, trigger "HMI_DB_Messages_Crane_wMessageWord2" bit 15
   803: 'Помилка енкодеру візка 4BR1', class MessageCrane, trigger "HMI_DB_Messages_Crane_wMessageWord3" bit 0
   804: 'Енкодер візка 4BR1 працює без помилок', class MessageCrane, trigger "HMI_DB_Messages_Crane_wMessageWord3" bit 1
   805: 'Помилка енкодеру візка 4BR2', class MessageCrane, trigger "HMI_DB_Messages_Crane_wMessageWord3" bit 2
   806: 'Енкодер візка 4BR2 працює без помилок', class MessageCrane, trigger "HMI_DB_Messages_Crane_wMessageWord3" bit 3
   807: 'Дозвіл роб. з будь-якої сторони від колони дозволено', class MessageCrane, trigger "HMI_DB_Messages_Crane_wMessageWord3" bit 4
   808: 'Дозвіл роб. з будь-якої сторони від колони заборонено', class MessageCrane, trigger "HMI_DB_Messages_Crane_wMessageWord3" bit 5
   784: 'Аварійний стоп', class ErrorCrane, trigger "HMI_DB_Alarms_Crane_AlarmWord1" bit 0
   785: 'Головний контактор вимкнений під час роботи', class ErrorCrane, trigger "HMI_DB_Alarms_Crane_AlarmWord1" bit 1
   802: 'Перегрів гальмівного резистора моста 4BT1', class ErrorCrane, trigger "HMI_DB_Alarms_Crane_AlarmWord1" bit 2
   811: 'Перегрів гальмівного резистора моста 4BT2', class ErrorCrane, trigger "HMI_DB_Alarms_Crane_AlarmWord1" bit 3
   812: 'Перегрів двигуна моста 4M1 (4KT1)', class ErrorCrane, trigger "HMI_DB_Alarms_Crane_AlarmWord1" bit 4
   813: 'Перегрів двигуна моста 4M2 (4KT2)', class ErrorCrane, trigger "HMI_DB_Alarms_Crane_AlarmWord1" bit 5
   814: 'Несправність частотного перетворювача 4UZ1', class ErrorCrane, trigger "HMI_DB_Alarms_Crane_AlarmWord1" bit 6
   815: 'Несправність частотного перетворювача 4UZ2', class ErrorCrane, trigger "HMI_DB_Alarms_Crane_AlarmWord1" bit 7
   816: 'Несправність енкодера 4BR1', class ErrorCrane, trigger "HMI_DB_Alarms_Crane_AlarmWord1" bit 8
   817: 'Несправність енкодера 4BR2', class ErrorCrane, trigger "HMI_DB_Alarms_Crane_AlarmWord1" bit 9
   818: 'Перевищення номінального вантажу крану (ОВП)', class ErrorCrane, trigger "HMI_DB_Alarms_Crane_AlarmWord1" bit 10
   819: 'Динамічний перекіс по швид. двигунів (Розбіжність > 150 об/хв під час ходу)', class ErrorCrane, trigger "HMI_DB_Alarms_Crane_AlarmWord1" bit 11
   820: 'Критичний статичний перекіс моста по датчиках енкодерів у міліметрах', class ErrorCrane, trigger "HMI_DB_Alarms_Crane_AlarmWord1" bit 12
   17: 'Перевищення номінального вантажу крану (ОВП)', class ErrorTrolley, trigger "HMI_DB_Alarms_Trolley_AlarmWord1" bit 6
   34: 'Контактор. вкл. роб. гальма. підйому 1KM1. Змінено стан з вимкн. на увімкн.', class MessageLiftUp, trigger "HMI_DB_Messages_LiftUp_wMessageWord3" bit 14
   55: 'Контактор. вкл. роб. гальма. підйому 1KM1. Змінено стан з увімкн. на вимкн.', class MessageLiftUp, trigger "HMI_DB_Messages_LiftUp_wMessageWord3" bit 15
   72: 'Контактор. вкл. вбуд. гальма. підйому 1KM2. Змінено стан з вимкн. на увімкн.', class MessageLiftUp, trigger "HMI_DB_Messages_LiftUp_wMessageWord4" bit 0
   73: 'Контактор. вкл. вбуд. гальма. підйому 1KM2. Змінено стан з увімкн. на вимкн.', class MessageLiftUp, trigger "HMI_DB_Messages_LiftUp_wMessageWord4" bit 1
   90: 'Контактор. вкл. аварій. гальма. підйому 1KM3. Змінено стан з вимкн. на увімкн.', class MessageLiftUp, trigger "HMI_DB_Messages_LiftUp_wMessageWord4" bit 2
   403: 'Контактор. вкл. аварій. гальма. підйому 1KM3. Змінено стан з увімкн. на вимкн.', class MessageLiftUp, trigger "HMI_DB_Messages_LiftUp_wMessageWord4" bit 3
   404: 'Контактор. вкл. роб. гальма. візка 3KM1. Змінено стан з вимкн. на увімкн.', class MessageTrolley, trigger "HMI_DB_Messages_Trolley_wMessageWord2" bit 10
   405: 'Контактор. вкл. роб. гальма. візка 3KM1. Змінено стан з увімкн. на вимкн.', class MessageTrolley, trigger "HMI_DB_Messages_Trolley_wMessageWord2" bit 11
   406: 'Контактор. вкл. роб. гальма. крану 4KM1. Змінено стан з вимкн. на увімкн.', class MessageCrane, trigger "HMI_DB_Messages_Crane_wMessageWord3" bit 6
   407: 'Контактор. вкл. роб. гальма. крану 4KM1. Змінено стан з увімкн. на вимкн.', class MessageCrane, trigger "HMI_DB_Messages_Crane_wMessageWord3" bit 7
   408: 'Реле дозволу вкл. лін. контактору 6K1. Змінено стан з вимкн. на увімкн.', class MessageContactor, trigger "HMI_DB_Messages_LinearContactor_wMessageWord4" bit 14
   409: 'Реле дозволу вкл. лін. контактору 6K1. Змінено стан з увімкн. на вимкн.', class MessageContactor, trigger "HMI_DB_Messages_LinearContactor_wMessageWord4" bit 15
   410: 'Реле вимкнення лін. контактору 6K2. Змінено стан з вимкн. на увімкн.', class MessageContactor, trigger "HMI_DB_Messages_LinearContactor_wMessageWord5" bit 0
   411: 'Реле вимкнення лін. контактору 6K2. Змінено стан з увімкн. на вимкн.', class MessageContactor, trigger "HMI_DB_Messages_LinearContactor_wMessageWord5" bit 1
   412: 'Реле включення дзвінка 9K1. Змінено стан з вимкн. на увімкн.', class MessageContactor, trigger "HMI_DB_Messages_LinearContactor_wMessageWord5" bit 2
   414: 'Реле включення дзвінка 9K2. Змінено стан з увімкн. на вимкн.', class MessageContactor, trigger "HMI_DB_Messages_LinearContactor_wMessageWord5" bit 3
   415: 'ПЛК працює без помилок', class MessageDiag, trigger "HMI_DB_Messages_Diag_wMessageWord1" bit 0
   416: 'Помилка ПЛК', class MessageDiag, trigger "HMI_DB_Messages_Diag_wMessageWord1" bit 1
   417: 'Модуль А1.2 працює нормально', class MessageDiag, trigger "HMI_DB_Messages_Diag_wMessageWord1" bit 2
   418: 'Модуль А1.2 вийшов з ладу', class MessageDiag, trigger "HMI_DB_Messages_Diag_wMessageWord1" bit 3
   419: 'Модуль А1.3 працює нормально', class MessageDiag, trigger "HMI_DB_Messages_Diag_wMessageWord1" bit 4
   420: 'Модуль А1.3 вийшов з ладу', class MessageDiag, trigger "HMI_DB_Messages_Diag_wMessageWord1" bit 5
   421: 'Модуль А1.4 працює нормально', class MessageDiag, trigger "HMI_DB_Messages_Diag_wMessageWord1" bit 6
   422: 'Модуль А1.4 вийшов з ладу', class MessageDiag, trigger "HMI_DB_Messages_Diag_wMessageWord1" bit 7
   423: 'Модуль А1.5 працює нормально', class MessageDiag, trigger "HMI_DB_Messages_Diag_wMessageWord1" bit 8
   424: 'Модуль А1.5 вийшов з ладу', class MessageDiag, trigger "HMI_DB_Messages_Diag_wMessageWord1" bit 9
   425: 'Scalance працює нормально', class MessageDiag, trigger "HMI_DB_Messages_Diag_wMessageWord1" bit 10
   426: 'Scalance вийшов з ладу', class MessageDiag, trigger "HMI_DB_Messages_Diag_wMessageWord1" bit 11
   427: 'Модуль CU працює нормально', class MessageDiag, trigger "HMI_DB_Messages_Diag_wMessageWord1" bit 12
   428: 'Модуль CU вийшов з ладу', class MessageDiag, trigger "HMI_DB_Messages_Diag_wMessageWord1" bit 13
   429: 'Зв'язок з ПЧ 1UZ1 у нормі', class MessageDiag, trigger "HMI_DB_Messages_Diag_wMessageWord1" bit 14
   431: 'Зв'язок з ПЧ 1UZ1 порушено', class MessageDiag, trigger "HMI_DB_Messages_Diag_wMessageWord1" bit 15
   433: 'Зв'язок з ПЧ 3UZ1 у нормі', class MessageDiag, trigger "HMI_DB_Messages_Diag_wMessageWord2" bit 0
   434: 'Зв'язок з ПЧ 3UZ1 порушено', class MessageDiag, trigger "HMI_DB_Messages_Diag_wMessageWord2" bit 1
   436: 'Зв'язок з ПЧ 4UZ1 у нормі', class MessageDiag, trigger "HMI_DB_Messages_Diag_wMessageWord2" bit 2
   437: 'Зв'язок з ПЧ 4UZ1 порушено', class MessageDiag, trigger "HMI_DB_Messages_Diag_wMessageWord2" bit 3
   438: 'Зв'язок з ПЧ 4UZ2 у нормі', class MessageDiag, trigger "HMI_DB_Messages_Diag_wMessageWord2" bit 4
   439: 'Зв'язок з ПЧ 4UZ2 порушено', class MessageDiag, trigger "HMI_DB_Messages_Diag_wMessageWord2" bit 5
   440: 'Зв'язок з енкодером 1BR у нормі', class MessageDiag, trigger "HMI_DB_Messages_Diag_wMessageWord2" bit 6
   441: 'Зв'язок з енкодером 1BR порушено', class MessageDiag, trigger "HMI_DB_Messages_Diag_wMessageWord2" bit 7
   442: 'Зв'язок з енкодером 3BR у нормі', class MessageDiag, trigger "HMI_DB_Messages_Diag_wMessageWord2" bit 8
   443: 'Зв'язок з енкодером 3BR порушено', class MessageDiag, trigger "HMI_DB_Messages_Diag_wMessageWord2" bit 9
   444: 'Зв'язок з енкодером 4BR1 у нормі', class MessageDiag, trigger "HMI_DB_Messages_Diag_wMessageWord2" bit 10
   445: 'Зв'язок з енкодером 4BR1 порушено', class MessageDiag, trigger "HMI_DB_Messages_Diag_wMessageWord2" bit 11
   446: 'Зв'язок з енкодером 4BR2 у нормі', class MessageDiag, trigger "HMI_DB_Messages_Diag_wMessageWord2" bit 12
   448: 'Зв'язок з енкодером 4BR2 порушено', class MessageDiag, trigger "HMI_DB_Messages_Diag_wMessageWord2" bit 13
   449: 'Автомат. вим. 9QF3. Змінено стан з вимкн. на увімкн.', class MessageSelf, trigger "HMI_DB_Messages_Self_wMessageWord1" bit 0
   450: 'Автомат. вим. 9QF3. Змінено стан з увімкн. на вимкн.', class MessageSelf, trigger "HMI_DB_Messages_Self_wMessageWord1" bit 1
   432: 'Автомат. вим. 9QF2. Змінено стан з вимкн. на увімкн.', class MessageSelf, trigger "HMI_DB_Messages_Self_wMessageWord1" bit 2
   435: 'Автомат. вим. 9QF2. Змінено стан з увімкн. на вимкн.', class MessageSelf, trigger "HMI_DB_Messages_Self_wMessageWord1" bit 3
   451: 'Софт. кінц. вимик. зупин мех. підйому у верхній точці у нормі', class MessageLiftUp, trigger "HMI_DB_Messages_LiftUp_wMessageWord4" bit 4
   452: 'Спрацював софт. кінц. вимик. зупин мех. підйому у верхній точці', class MessageLiftUp, trigger "HMI_DB_Messages_LiftUp_wMessageWord4" bit 5
   453: 'Софт. кінц. вимик. зупин мех. підйому у нижній точці у нормі', class MessageLiftUp, trigger "HMI_DB_Messages_LiftUp_wMessageWord4" bit 6
   454: 'Спрацював софт. кінц. вимик. зупин мех. підйому у нижній точці', class MessageLiftUp, trigger "HMI_DB_Messages_LiftUp_wMessageWord4" bit 7
   455: 'Софт. кінц. вимик. зупин мех. візка попереду у нормі', class MessageTrolley, trigger "HMI_DB_Messages_Trolley_wMessageWord2" bit 12
   456: 'Спрацював софт. кінц. вимик. зупин мех. візка попереду', class MessageTrolley, trigger "HMI_DB_Messages_Trolley_wMessageWord2" bit 13
   457: 'Софт. кінц. вимик. зупин мех. візка позаду у нормі', class MessageTrolley, trigger "HMI_DB_Messages_Trolley_wMessageWord2" bit 14
   458: 'Спрацював софт. кінц. вимик. зупин мех. візка позаду', class MessageTrolley, trigger "HMI_DB_Messages_Trolley_wMessageWord2" bit 15
   459: 'Софт. кінц. вимик. зупин мех. моста зправа у нормі', class MessageCrane, trigger "HMI_DB_Messages_Crane_wMessageWord3" bit 8
   460: 'Спрацював софт. кінц. вимик. зупин мех. моста зправа', class MessageCrane, trigger "HMI_DB_Messages_Crane_wMessageWord3" bit 9
   461: 'Софт. кінц. вимик. зупин мех. моста зліва у нормі', class MessageCrane, trigger "HMI_DB_Messages_Crane_wMessageWord3" bit 10
   462: 'Спрацював софт. кінц. вимик. зупин мех. моста зліва', class MessageCrane, trigger "HMI_DB_Messages_Crane_wMessageWord3" bit 11
   471: 'Зв'язок з енкодером 3BR порушено', class ErrorDiag, trigger "HMI_DB_Alarms_Diagn_AlarmWord1" bit 7
   466: 'Зв'язок з модулем А1.3 порушено', class ErrorDiag, trigger "HMI_DB_Alarms_Diagn_AlarmWord1" bit 2
   467: 'Зв'язок з модулем А1.4 порушено', class ErrorDiag, trigger "HMI_DB_Alarms_Diagn_AlarmWord1" bit 3
   468: 'Зв'язок з модулем А1.5 порушено', class ErrorDiag, trigger "HMI_DB_Alarms_Diagn_AlarmWord1" bit 4
   469: 'Зв'язок з модулем А1.6 порушено', class ErrorDiag, trigger "HMI_DB_Alarms_Diagn_AlarmWord1" bit 5
   463: 'Зв'язок з модулем ПЛК порушено', class ErrorDiag, trigger "HMI_DB_Alarms_Diagn_AlarmWord1" bit 0
   465: 'Зв'язок з модулем А1.2 порушено', class ErrorDiag, trigger "HMI_DB_Alarms_Diagn_AlarmWord1" bit 1
   472: 'Зв'язок з енкодером 4BR1 порушено', class ErrorDiag, trigger "HMI_DB_Alarms_Diagn_AlarmWord1" bit 8
   473: 'Зв'язок з енкодером 4BR2 порушено', class ErrorDiag, trigger "HMI_DB_Alarms_Diagn_AlarmWord1" bit 9
   474: 'Зв'язок з модулем U1 порушено', class ErrorDiag, trigger "HMI_DB_Alarms_Diagn_AlarmWord1" bit 10
   475: 'Зв'язок з ПЧ 1UZ1 порушено', class ErrorDiag, trigger "HMI_DB_Alarms_Diagn_AlarmWord1" bit 11
   476: 'Зв'язок з ПЧ 3UZ1 порушено', class ErrorDiag, trigger "HMI_DB_Alarms_Diagn_AlarmWord1" bit 12
   477: 'Зв'язок з ПЧ 4UZ1 порушено', class ErrorDiag, trigger "HMI_DB_Alarms_Diagn_AlarmWord1" bit 13
   478: 'Зв'язок з ПЧ 4UZ2 порушено', class ErrorDiag, trigger "HMI_DB_Alarms_Diagn_AlarmWord1" bit 14
   470: 'Зв'язок з енкодером 1BR порушено', class ErrorDiag, trigger "HMI_DB_Alarms_Diagn_AlarmWord1" bit 6
   485: 'Мех. підйому не калібровано', class ErrorLiftUp, trigger "HMI_DB_Alarms_LiftUp_AlarmWord2" bit 5
   491: 'Мех. візка не калібровано', class ErrorTrolley, trigger "HMI_DB_Alarms_Trolley_AlarmWord2" bit 5
   498: 'Мех. крану не калібровано', class ErrorCrane, trigger "HMI_DB_Alarms_Crane_AlarmWord2" bit 5
   504: 'Обмеження рузу назад візка у межах колони', class ErrorContactor, trigger "HMI_DB_Alarms_Contactor_AlarmWord2" bit 11
   505: 'Спрацювала пожежна сигналізація', class ErrorContactor, trigger "HMI_DB_Alarms_Contactor_AlarmWord2" bit 12
   506: 'Значення енкодера 4BR1 після увімк. не узгоджено', class CraneCalibrDiag, trigger "HMI_DB_Warnings_Crane" bit 0
   492: 'Значення енкодера 4BR1 змінилось без команди на рух', class CraneCalibrDiag, trigger "HMI_DB_Warnings_Crane" bit 1
   493: 'Значення енкодера 4BR1 змінилось без актив. ручн. приводу', class CraneCalibrDiag, trigger "HMI_DB_Warnings_Crane" bit 2
   494: 'Значення енкодера 4BR1 не змінюється після початку руху', class CraneCalibrDiag, trigger "HMI_DB_Warnings_Crane" bit 3
   495: 'Фізична зміна енкодера 4BR1', class CraneCalibrDiag, trigger "HMI_DB_Warnings_Crane" bit 4
   497: 'Значення енкодера 4BR2 після увімк. не узгоджено', class CraneCalibrDiag, trigger "HMI_DB_Warnings_Crane" bit 6
   499: 'Значення енкодера 4BR2 змінилось без команди на рух', class CraneCalibrDiag, trigger "HMI_DB_Warnings_Crane" bit 7
   500: 'Значення енкодера 4BR2 змінилось без актив. ручн. приводу', class CraneCalibrDiag, trigger "HMI_DB_Warnings_Crane" bit 8
   501: 'Значення енкодера 4BR2 не змінюється після початку руху', class CraneCalibrDiag, trigger "HMI_DB_Warnings_Crane" bit 9
   502: 'Фізична зміна енкодера 4BR2', class CraneCalibrDiag, trigger "HMI_DB_Warnings_Crane" bit 10
   503: 'Положення мех. підйому після увімк. не узгоджено', class LiftUpCalibrDiag, trigger "HMI_DB_Warnings_LiftUp" bit 0
   480: 'Положення мех. пійдому змінилось без актив. ручн. приводу', class LiftUpCalibrDiag, trigger "HMI_DB_Warnings_LiftUp" bit 1
   481: 'Положення мех. пійдому змінилось без актив. ручн. приводу', class LiftUpCalibrDiag, trigger "HMI_DB_Warnings_LiftUp" bit 2
   507: 'Положення мех. пійдому не змінюється після початку руху', class LiftUpCalibrDiag, trigger "HMI_DB_Warnings_LiftUp" bit 3
   482: 'Фізична зміна енкодера мех. підйому', class LiftUpCalibrDiag, trigger "HMI_DB_Warnings_LiftUp" bit 4
   483: 'Положення мех. візка після увімк. не узгоджено', class TrolleyCalibrDiag, trigger "HMI_DB_Warnings_Trolley" bit 0
   484: 'Положення мех. візка змінилось без команди на рух', class TrolleyCalibrDiag, trigger "HMI_DB_Warnings_Trolley" bit 1
   486: 'Положення мех. візка змінилось без актив. ручн. приводу', class TrolleyCalibrDiag, trigger "HMI_DB_Warnings_Trolley" bit 2
   487: 'Положення мех. візка не змінюється після початку руху', class TrolleyCalibrDiag, trigger "HMI_DB_Warnings_Trolley" bit 3
   488: 'Фізична зміна енкодера мех.візка', class TrolleyCalibrDiag, trigger "HMI_DB_Warnings_Trolley" bit 4
   489: 'Порушено топологію кільця', class ErrorDiag, trigger "HMI_DB_Alarms_Diagn_AlarmWord1" bit 15

